// TIA Portal project "GridTest2093" (V19)

(* hardware
DEVICE "S7-1200 station_1"  S7-1200 Station
   slot 0: "Rack_0"  S7-1200 Rack  Rack  V1.0
   slot 1: "PLC_1"  CPU 1214C DC/DC/DC  6ES7 214-1AG40-0XB0  V4.6
   slot 2: "AI 4x13BIT_1"  6ES7 231-4HD32-0XB0  V2.1
   slot 3: "AI 8x13BIT_1"  6ES7 231-4HF32-0XB0  V2.1
   slot 4: "AQ 4x14BIT_1"  6ES7 232-4HD32-0XB0  V2.1
   slot 5: "DQ 8x24VDC _1"  SM 1222 DQ8 x 24VDC  6ES7 222-1BF32-0XB0  V2.0
*)

// ===== PLC "PLC_1"  CPU 1214C DC/DC/DC =====

VAR_GLOBAL   // PLC tag table "Default tag table"
   "test1" AT %Q0.0 : Bool;
   "test2" AT %Q0.1 : Bool;
END_VAR

VAR_GLOBAL   // PLC tag table "Grid"
   "o_G1_Inverter_ON" AT %Q0.2 : Bool;
   "o_G1_KV_ON" AT %Q0.3 : Bool;
   "o_G2_Inverter_ON" AT %Q0.4 : Bool;
   "o_G2_KV_ON" AT %Q0.5 : Bool;
   "ao_G1_KV_SET" AT %QW112 : Int;
   "ao_G2_KV_SET" AT %QW114 : Int;
   "ai_G1_KVFB" AT %IW96 : Int;
   "ai_G2_KVFB" AT %IW98 : Int;
END_VAR

VAR_GLOBAL   // PLC tag table "remVals"
   "ai_remKVrdg" AT %IW112 : Int;
   "ai_remMArdg" AT %IW114 : Int;
   "ai_remIfrdg" AT %IW116 : Int;
   "i_remProcOK" AT %I0.0 : Bool;
   "i_rem_NotUsed" AT %I0.1 : Bool;
   "i_cam_EXPOSE_OK" AT %I0.2 : Bool;
   "o_GoRemote" AT %Q20.0 : Bool;
   "o_remSmall" AT %Q20.1 : Bool;
   "o_remHiSpd" AT %Q20.2 : Bool;
   "o_remNotUsed" AT %Q20.3 : Bool;
   "o_Sonalert" AT %Q20.4 : Bool;
   "o_cam_SHORT_SYNC" AT %Q20.5 : Bool;
   "o_cam_LONG_SYNC" AT %Q20.6 : Bool;
   "ao_KVSP" AT %QW116 : Int;
END_VAR

DATA_BLOCK "Inputs_DB"   // DB9
{ S7_Optimized_Access := 'TRUE' }
VERSION : 0.1
// stored: InstanceOfName Inputs
"Inputs"
BEGIN
END_DATA_BLOCK

DATA_BLOCK "Step_Values_DB"   // DB16
{ S7_Optimized_Access := 'TRUE' }
VERSION : 0.1
// stored: InstanceOfName Step_Values
"Step_Values"
BEGIN
END_DATA_BLOCK

DATA_BLOCK "Outputs_DB"   // DB17
{ S7_Optimized_Access := 'TRUE' }
VERSION : 0.1
// stored: InstanceOfName Outputs
"Outputs"
BEGIN
END_DATA_BLOCK

DATA_BLOCK "Run_Sched_DB"   // DB37
{ S7_Optimized_Access := 'TRUE' }
VERSION : 0.1
// stored: InstanceOfName Run_Sched
"Run_Sched"
BEGIN
END_DATA_BLOCK

DATA_BLOCK "ALARMS_CHECK_DB"   // DB38
{ S7_Optimized_Access := 'TRUE' }
VERSION : 0.1
// stored: InstanceOfName ALARMS_CHECK
"ALARMS_CHECK"
BEGIN
END_DATA_BLOCK

DATA_BLOCK "Reset_DB"   // DB41
{ S7_Optimized_Access := 'TRUE' }
VERSION : 0.1
// stored: InstanceOfName Reset
"Reset"
BEGIN
END_DATA_BLOCK

DATA_BLOCK "Heat_Int_DB"   // DB42
{ S7_Optimized_Access := 'TRUE' }
VERSION : 0.1
// stored: InstanceOfName Heat_Int
"Heat_Int"
BEGIN
END_DATA_BLOCK

DATA_BLOCK "Retests_DB"   // DB43
{ S7_Optimized_Access := 'TRUE' }
VERSION : 0.1
// stored: InstanceOfName Retests
"Retests"
BEGIN
END_DATA_BLOCK

// folder: Datablocks

DATA_BLOCK "LVtest"   // DB1
{ S7_Optimized_Access := 'FALSE' }
VERSION : 0.1
   VAR
      val1 : Bool := false;
      val2 : Bool;
      num1 : DInt := 10;
      str1 : String := 'hello';
      val3 : Bool := false;
      str2 : String := 'nice';
      val4 : Bool;
      steptest : Int;
   END_VAR
BEGIN
END_DATA_BLOCK

DATA_BLOCK "BIASDIFF"   // DB3
{ S7_Optimized_Access := 'FALSE' }
VERSION : 0.1
   VAR
      BIAS_ZERO : Bool;
      DIFF_ZERO : Bool;
      BIAS : Real;
      DIFF : Real;
      BIAS_DIFF_OK : Bool;
      BIAS_RSE : Bool;
      BIAS_LWR : Bool;
      DIFF_RSE : Bool;
      DIFF_LWR : Bool;
      Max_DIFF : Real;
      Min_DIFF : Real;
      DIFF_TOGGLE : Bool;
      BIAS_DIFF_TMR : Time;
      BIAS_Prior : Real;
      DIFF_Prior : Real;
      delta_BIAS : Real;
   END_VAR
BEGIN
END_DATA_BLOCK

DATA_BLOCK "Gx"   // DB4
{ S7_Optimized_Access := 'FALSE' }
VERSION : 0.1
   VAR
      max_Gx : Real;
      min_Gx : Real;
      G1V_SP : Real;
      G2V_SP : Real;
      schd_max_Gx : Array[0..2] of Real;
      G1Invert : Bool;   // G1 Invert output
      G1KVOn : Bool;   // G1 KV enable output
      G1KVSet : Real;   // G1 KV set output
      G2Invert : Bool;   // G2 Invert output
      G2KVON : Bool;   // G2 KV enable output
      G2KVSet : Real;   // G2 KV set output
      G1KVfb : DInt;   // G1 KV feedback input
      G2KVfb : DInt;   // G2 KV feedback input
      Gx_LIMIT : Real;
   END_VAR
BEGIN
END_DATA_BLOCK

DATA_BLOCK "Params"   // DB5
{ S7_Optimized_Access := 'FALSE' }
VERSION : 0.1
   VAR
      stp_PARAMS : Array[0..31] of Bool;
      PARAMS : Array[0..31] of Bool;
      stp_TEST : Array[0..31] of Bool;
   END_VAR
BEGIN
END_DATA_BLOCK

DATA_BLOCK "Limits"   // DB6
{ S7_Optimized_Access := 'FALSE' }
VERSION : 0.1
   VAR
      LIMITS : Array[0..39] of Real;
      LIMITS_PB : Array[0..7] of Bool;
   END_VAR
BEGIN
   // LIMITS[0] : max GxV
   // LIMITS[1] : max GxuA
   // LIMITS[2] : max EfDr
   // LIMITS[3] : min EfDr
   // LIMITS[4] : max KV
   // LIMITS[5] : MA%HI Circ Brkr ABORT
   // LIMITS[6] : max MA ABORT
   // LIMITS[7] : GRID Comms bad mS ABORT
   // LIMITS[8] : max short pulse tries
   // LIMITS[9] : .....
   // LIMITS[10] : short EXP Cool delay mS to next
   // LIMITS[11] : mS rdg delay
   // LIMITS[12] : max Temp ABORT
   // LIMITS[13] : pulse MA OK%tol
   // LIMITS[14] : pulse If OK %tol
   // LIMITS[15] : ......
   // LIMITS[16] : EfDr delta max adj
   // LIMITS[17] : MA REG Gain
   // LIMITS[18] : If REG Gain
   // LIMITS[19] : Cutoff Test BIAS Gain
   // LIMITS[20] : If rdgs averaged
   // LIMITS[21] : MA rdgs avgd for Cutoff
   // LIMITS[22] : Xpos Offset mm
   // LIMITS[23] : Zpos Offset mm
   // LIMITS[24] : Ypos Offset mm
   // LIMITS[25] : .....
   // LIMITS[26] : .....
   // LIMITS[27] : DEFL adj Gain, V/mm LO
   // LIMITS[28] : .....
   // LIMITS[29] : Change Mode TD mS
   // LIMITS[30] : .....
   // LIMITS[31] : Heat/to TEMP params[1]
   // LIMITS[32] : Cool/to TEMP params[5]
   // LIMITS[35] : min -delta BIAS adj Width
   // LIMITS[39] : auto re-TEST # times
   // LIMITS[38] : MA REG Gain #2
   // LIMITS[37] : Width adj BIAS Gain (140KV)
   // LIMITS[36] : .....
   // LIMITS[34] : max +delta BIAS adj Width
   // LIMITS[33] : .....
   // LIMITS_PB[0] : NO GRID TANK
   // LIMITS_PB[1] : NO CAMERA
   // LIMITS_PB[2] : Cheat ProcNOK
   // LIMITS_PB[3] : SIM IO
   // LIMITS_PB[4] : store IMAGE
   // LIMITS_PB[5] : cycle Go User Sync
   // LIMITS_PB[6] : CAL (Remote = On)
   // LIMITS_PB[7] : Over Expose Alarm
END_DATA_BLOCK

DATA_BLOCK "Schd"   // DB7
{ S7_Optimized_Access := 'TRUE' }
VERSION : 0.1
   VAR
      RUN : Bool;
   END_VAR
BEGIN
END_DATA_BLOCK

DATA_BLOCK "ANALOG_IO"   // DB8
{ S7_Optimized_Access := 'FALSE' }
VERSION : 0.1
   VAR
      remKVSP : Real := 0.0;
      remKVrdg : Real := 0.0;
      remMASP : Real := 0.0;
      remMArdg : Real := 0.0;
      remEfDrSP : Real := 0.0;
      remEfDrRdg : Real := 0.0;
      remIfrdg : Real := 0.0;
      G1V_SP : Real := 0.0;
      G2V_SP : Real := 0.0;
      G1RDG : Real := 0.0;
      G2RDG : Real := 0.0;
   END_VAR
BEGIN
END_DATA_BLOCK

DATA_BLOCK "Schedule"   // DB10
{ S7_Optimized_Access := 'FALSE' }
VERSION : 0.1
   VAR
      PARAMS : Array[0..31] of Real;
      KV : Array[0..31] of Real;
      MAIF : Array[0..31] of Real;
      EXPtime : Array[0..31] of Real;
      COOLtime : Array[0..31] of Real;
      scansMode : Array[0..31] of Real;
      dataitem : Array[0..31] of Real;
      min : Array[0..31] of Real;
      max : Array[0..31] of Real;
      initBIAS : Array[0..31] of Real;
      initDIFF : Array[0..31] of Real;
      maxGx : Array[0..31] of Real;
      initEfDr : Array[0..31] of Real;
      maxTries : Array[0..31] of Real;
      TEST : Array[0..31] of Real;
      LIM1 : Array[0..31] of Real;
      LIM2 : Array[0..31] of Real;
      LIM3 : Array[0..31] of Real;
      LIM4 : Array[0..31] of Real;
   END_VAR
BEGIN
END_DATA_BLOCK

DATA_BLOCK "DIGITAL_IO"   // DB11
{ S7_Optimized_Access := 'FALSE' }
VERSION : 0.1
   VAR
      GORemote : Bool;
      remSMALL : Bool;
      remHiSpd : Bool;
      Sonalert : Bool;
      cam_SHORT_SYNC : Bool;
      cam_LONG_SYNC : Bool;
      remProcOK : Bool;
      cam_EXPOSURE_OK : Bool;
      G1V_Invert : Bool;
      G1V_On : Bool;
      G2V_Invert : Bool;
      G2V_On : Bool;
      SPARE1 : Bool;
      SPARE2 : Bool;
      SPARE3 : Bool;
      SPARE4 : Bool;
   END_VAR
BEGIN
END_DATA_BLOCK

DATA_BLOCK "OffsetGain"   // DB12
{ S7_Optimized_Access := 'FALSE' }
VERSION : 0.1
   VAR
      remKVSPOffset : Real;
      remKVSPGain : Real;
      remKVrdgOffset : Real;
      remKVrdgGain : Real;
      remMASPOffset : Real;
      remMASPGain : Real;
      remMArdgOffset : Real;
      remMArdgGain : Real;
      remEfDrSPOffset : Real;
      remEfDrSPGain : Real;
      remEfDrRdgOffset : Real;
      remEfDrRdgGain : Real;
      remIfRdgOffset : Real;
      remIfRdgGain : Real;
      G1V_SP_Offset : Real;
      G1V_SP_Gain : Real;
      G1V_RDG_Offset : Real;
      G1V_RDG_Gain : Real;
      G2V_SP_Offset : Real;
      G2V_SP_Gain : Real;
      G2V_RDG_Offset : Real;
      G2V_RDG_Gain : Real;
   END_VAR
BEGIN
END_DATA_BLOCK

DATA_BLOCK "Tube"   // DB13
{ S7_Optimized_Access := 'FALSE' }
VERSION : 0.1
   VAR
      RTC : Real;
      HS : Real;
      T100 : Real;
      T0 : Real;
      AP : Real;
   END_VAR
BEGIN
END_DATA_BLOCK

DATA_BLOCK "Run_Control"   // DB14
{ S7_Optimized_Access := 'FALSE' }
VERSION : 0.1
   VAR
      First_Step : Int;
      Final_Step : Int;
      Current_Step : Int;
      Run : Int;
      Reset : Int;
      GoRemote : Int;
   END_VAR
BEGIN
END_DATA_BLOCK

DATA_BLOCK "Alarms"   // DB15
{ S7_Optimized_Access := 'FALSE' }
VERSION : 0.1
   VAR
      Alarms : Array[0..31] of Bool;
      Alarm_Clear : Bool;
      buff1 : Int;
      ProcNOK_Clear : Bool;
      buff2 : Int;
      ALARM_ACTIVE : Bool;
      PROCNOK_ACTIVE : Bool;
   END_VAR
BEGIN
   // Alarms[0] : COMMS ERROR
   // Alarms[1] : RUN LOG OPEN >> CLOSE
   // Alarms[2] : remProcNOK 50 sec
   // Alarms[3] : expose NOK 90 sec
   // Alarms[4] : exp NOK 5min >> ABORT
   // Alarms[5] : GRID COMMS >> ABORT
   // Alarms[6] : MA HI >> ABORT
   // Alarms[7] : max tries LIM[9] >> ABORT
   // Alarms[8] : ProcNOK 90 sec
   // Alarms[9] : ProcNOK CHEATED (LIM)
   // Alarms[10] : Gx Volts HI/LO
   // Alarms[11] : TEMP HI LIM[13] >> ABORT
   // Alarms[12] : Cam User Sync <> 2 15 sec
   // Alarms[13] : CLOSE DATA SHEET LOG
   // Alarms[14] : Gx uA > LIM[2] >> ABORT
   // Alarms[15] : EXPOSE LONG >> ABORT
   // Alarms[31] : DONE
END_DATA_BLOCK

DATA_BLOCK "Cam"   // DB18
{ S7_Optimized_Access := 'FALSE' }
VERSION : 0.1
   VAR
      X_defl : Real;
      Z_defl : Real;
      Y_defl : Real;
      cam_Wref : Real;
      cam_Lref : Real;
      cam_Xref : Real;
      cam_Zref : Real;
      cam_Yref : Real;
      cam_WIDTH : Real;
      cam_LENGTH : Real;
      cam_Xpos : Real;
      cam_Zpos : Real;
      cam_Ypos : Real;
      cam_MAG : Real;
      cam_FRAME_RATE : Real;
      image_KV : Real;
      image_MA : Real;
      image_G1 : Real;
      image_G2 : Real;
      image_BIAS : Real;
      image_DIFF : Real;
      cam_POS : Real;
      cam_USER_SYNC : Int;
      cam_DATA : Int;
      BIAS_ref : Int;
      cam_PEAK : Int;
      cam_OB_pk : Int;
      cam_Mode : Int;
      cam_PERCENT_MAX : Int;
      NO_CAMERA : Bool;
      IMAGE_ACQUIRED : Bool;
      STORE_IMAGE : Bool;
      cam_CAL_OFFSET : Bool;
      cam_STATUS : String;
      cam_IMAGE_PATH : String;
   END_VAR
BEGIN
END_DATA_BLOCK

DATA_BLOCK "pulse"   // DB19
{ S7_Optimized_Access := 'TRUE' }
VERSION : 0.1
   VAR
      pulse_KV : Int;
      pulse_MA : Int;
      pulse_If : Int;
      pulse_EfDr : Int;
      pulse_G2 : Int;
      pulse_G1 : Int;
      shortpulse_tries : Int;
      XPOSE_SEC : Int;
      COOL_SEC : Int;
      rdgs_avgd : Int;
      shortpulsetmr : Time;
      pulsePeriod : Real;
   END_VAR
BEGIN
END_DATA_BLOCK

DATA_BLOCK "ref"   // DB20
{ S7_Optimized_Access := 'TRUE' }
VERSION : 0.1
   VAR
      EfDr_ref : Real;
      BIAS_ref : Real;
   END_VAR
BEGIN
END_DATA_BLOCK

DATA_BLOCK "Prior"   // DB21
{ S7_Optimized_Access := 'TRUE' }
VERSION : 0.1
   VAR
      BIAS_Prior : Real;
      DIFF_Prior : Real;
      EfDr_Prior : Real;
   END_VAR
BEGIN
END_DATA_BLOCK

DATA_BLOCK "Results"   // DB22
{ S7_Optimized_Access := 'FALSE' }
VERSION : 0.1
   VAR
      testVAL : Real;
      min : Real;
      max : Real;
      KV : Real;
      MA : Real;
      EfDr : Real;
      "If" : Real;
      Temp : Real;
      G1V : Real;
      G2V : Real;
      Width : Real;
      Length : Real;
      Xdefl : Real;
      Zdefl : Real;
      Ydefl : Real;
      Xpos : Real;
      Zpos : Real;
      Ypos : Real;
      Mag : Real;
      pk : Real;
      OBpk : Real;
      tries : Real;
      scansmode : Real;
      dataitem : Real;
      Pass_Fail : Int;
   END_VAR
BEGIN
END_DATA_BLOCK

DATA_BLOCK "Chain_Schedule"   // DB23
{ S7_Optimized_Access := 'TRUE' }
VERSION : 0.1
   VAR
      Params : Real;
      KV : Real;
      MAIf : Real;
      EXPtime : Real;
      COOLtime : Real;
      scansMode : Real;
      dataitem : Real;
      min : Real;
      max : Real;
      initBIAS : Real;
      initDIFF : Real;
      maxGx : Real;
      initEfDr : Real;
      maxTries : Real;
      TEST : Real;
      LIM1 : Real;
      LIM2 : Real;
      LIM3 : Real;
      LIM4 : Real;
   END_VAR
BEGIN
END_DATA_BLOCK

DATA_BLOCK "System"   // DB24
{ S7_Optimized_Access := 'FALSE' }
VERSION : 0.1
   VAR
      COOLING : Bool;
      GoRemote : Bool;
      Temp_set : Real;
      Temp_rdg : Real;
      XPOSE_SEC : Real;
      RPTS : Int;
      Exp_MA_If_OK : Bool;
      Sleep : Bool;
   END_VAR
BEGIN
END_DATA_BLOCK

DATA_BLOCK "ProcOK"   // DB25
{ S7_Optimized_Access := 'FALSE' }
VERSION : 0.1
   VAR
      ProcOKArray : Array[0..31] of Bool;
      ProcOK : Bool;
   END_VAR
BEGIN
   ProcOKArray[0] := true;
   ProcOKArray[1] := true;
   ProcOKArray[2] := true;
   ProcOKArray[3] := true;
   ProcOKArray[4] := true;
   ProcOKArray[5] := true;
   ProcOKArray[6] := true;
   ProcOKArray[7] := true;
   ProcOKArray[8] := true;
   ProcOKArray[9] := true;
   ProcOKArray[10] := true;
   ProcOKArray[11] := true;
   ProcOKArray[12] := true;
   ProcOKArray[13] := true;
   ProcOKArray[14] := true;
   ProcOKArray[15] := true;
   ProcOKArray[16] := true;
   ProcOKArray[17] := true;
   ProcOKArray[18] := true;
   ProcOKArray[19] := true;
   ProcOKArray[20] := true;
   ProcOKArray[21] := true;
   ProcOKArray[22] := true;
   ProcOKArray[23] := true;
   ProcOKArray[24] := true;
   ProcOKArray[25] := true;
   ProcOKArray[26] := true;
   ProcOKArray[27] := true;
   ProcOKArray[28] := true;
   ProcOKArray[29] := true;
   ProcOKArray[30] := true;
   ProcOKArray[31] := true;
END_DATA_BLOCK

DATA_BLOCK "StepVals"   // DB26
{ S7_Optimized_Access := 'TRUE' }
VERSION : 0.1
   VAR
      PARAMS : Real;
      KV : Real;
      MAIf : Real;
      EXPtime : Real;
      COOLtime : Real;
      scansMode : Real;
      dataitem : Real;
      min : Real;
      max : Real;
      initBIAS : Real;
      initDIFF : Real;
      maxGx : Real;
      initEfDr : Real;
      maxTries : Real;
      TEST : Real;
      LIM1 : Real;
      LIM2 : Real;
      LIM3 : Real;
      LIM4 : Real;
   END_VAR
BEGIN
END_DATA_BLOCK

DATA_BLOCK "Misc"   // DB31
{ S7_Optimized_Access := 'FALSE' }
VERSION : 0.1
   VAR
      CutOff_avg_MA : Bool;
      rem_MA_rdg_avg : Real;
      Blinkingtme : Real;
   END_VAR
BEGIN
END_DATA_BLOCK

DATA_BLOCK "Cutoff"   // DB32
{ S7_Optimized_Access := 'TRUE' }
VERSION : 0.1
   VAR
      cutoff_BIAS : Real;
      cutoff_avg_MA : Bool;
   END_VAR
BEGIN
END_DATA_BLOCK

DATA_BLOCK "Remote"   // DB33
{ S7_Optimized_Access := 'TRUE' }
VERSION : 0.1
   VAR
      remEfDr_SP : Real;
   END_VAR
BEGIN
END_DATA_BLOCK

DATA_BLOCK "Cam(int)"   // DB34
{ S7_Optimized_Access := 'FALSE' }
VERSION : 0.1
   VAR
      cam_USER_SYNC : Int;
      cam_DATA : Int;
      BIAS_ref : Int;
      cam_PEAK : Int;
      cam_OB_pk : Int;
      cam_Mode : Int;
      cam_PERCENT_MAX : Int;
   END_VAR
BEGIN
END_DATA_BLOCK

DATA_BLOCK "Cam(bool)"   // DB35
{ S7_Optimized_Access := 'FALSE' }
VERSION : 0.1
   VAR
      NO_CAMERA : Bool;
      IMAGE_ACQUIRED : Bool;
      STORE_IMAGE : Bool;
      cam_CAL_OFFSET : Bool;
   END_VAR
BEGIN
END_DATA_BLOCK

DATA_BLOCK "Cam(string)"   // DB36
{ S7_Optimized_Access := 'FALSE' }
VERSION : 0.1
   VAR
      cam_STATUS : String;
      cam_IMAGE_PATH : String;
   END_VAR
BEGIN
END_DATA_BLOCK

DATA_BLOCK "Process"   // DB39
{ S7_Optimized_Access := 'FALSE' }
VERSION : 0.1
   VAR
      Run_Init : Bool;
      Step_Init : Bool := true;
      Running : Bool;
      Step_Running : Bool;
      Step_Done : Bool;
      Schedule_Done : Bool;
      Retest_Done : Bool;
      Results_Ready : Bool;
   END_VAR
BEGIN
END_DATA_BLOCK

DATA_BLOCK "Retest"   // DB40
{ S7_Optimized_Access := 'FALSE' }
VERSION : 0.1
   VAR
      Retest_Step : Int;
      Retest_End : Int;
      Retest_Type : Int;   // Retest=1: Retest Retest_Step only; Retest=2: Retest Retest_Step to End
      Retests : Int;
      Retries : Int;
      Retest : Bool;
   END_VAR
BEGIN
END_DATA_BLOCK

// folder: System blocks/Program resources

DATA_BLOCK "IEC_Timer_0_DB"   // DB2
{ S7_Optimized_Access := 'FALSE' }
AUTHOR : Simatic
FAMILY : IEC
NAME : IEC_TMR
VERSION : 1.0
// stored: InstanceOfName IEC_TIMER
"IEC_TIMER"
BEGIN
END_DATA_BLOCK

DATA_BLOCK "BIAS_Step_tmr1"   // DB27
{ S7_Optimized_Access := 'TRUE' }
AUTHOR : Simatic
FAMILY : IEC
NAME : IEC_TMR
VERSION : 1.0
// stored: InstanceOfName IEC_TIMER
"IEC_TIMER"
BEGIN
END_DATA_BLOCK

DATA_BLOCK "BIAS_Step_tmr2"   // DB28
{ S7_Optimized_Access := 'TRUE' }
AUTHOR : Simatic
FAMILY : IEC
NAME : IEC_TMR
VERSION : 1.0
// stored: InstanceOfName IEC_TIMER
"IEC_TIMER"
BEGIN
END_DATA_BLOCK

DATA_BLOCK "BIAS_Step_tmr3"   // DB29
{ S7_Optimized_Access := 'TRUE' }
AUTHOR : Simatic
FAMILY : IEC
NAME : IEC_TMR
VERSION : 1.0
// stored: InstanceOfName IEC_TIMER
"IEC_TIMER"
BEGIN
END_DATA_BLOCK

DATA_BLOCK "BIAS_Step_tmr4"   // DB30
{ S7_Optimized_Access := 'TRUE' }
AUTHOR : Simatic
FAMILY : IEC
NAME : IEC_TMR
VERSION : 1.0
// stored: InstanceOfName IEC_TIMER
"IEC_TIMER"
BEGIN
END_DATA_BLOCK

// folder: (top level)

ORGANIZATION_BLOCK "Main"   // OB1, LAD, ProgramCycle
TITLE = "Main Program Sweep (Cycle)"
{ S7_Optimized_Access := 'TRUE' }
VERSION : 0.1
   VAR_INPUT
      Initial_Call : Bool;   // Initial call of this OB
      Remanence : Bool;   // =True, if remanent data are available
   END_VAR
   VAR_TEMP
      test : Bool;
      "step" : Int;
      Blinkingtimer : Real;
   END_VAR
   VAR_TEMP   // added for the SCL form of the ladder/FBD networks
      _w1 : Bool;
   END_VAR
BEGIN

REGION Network 1
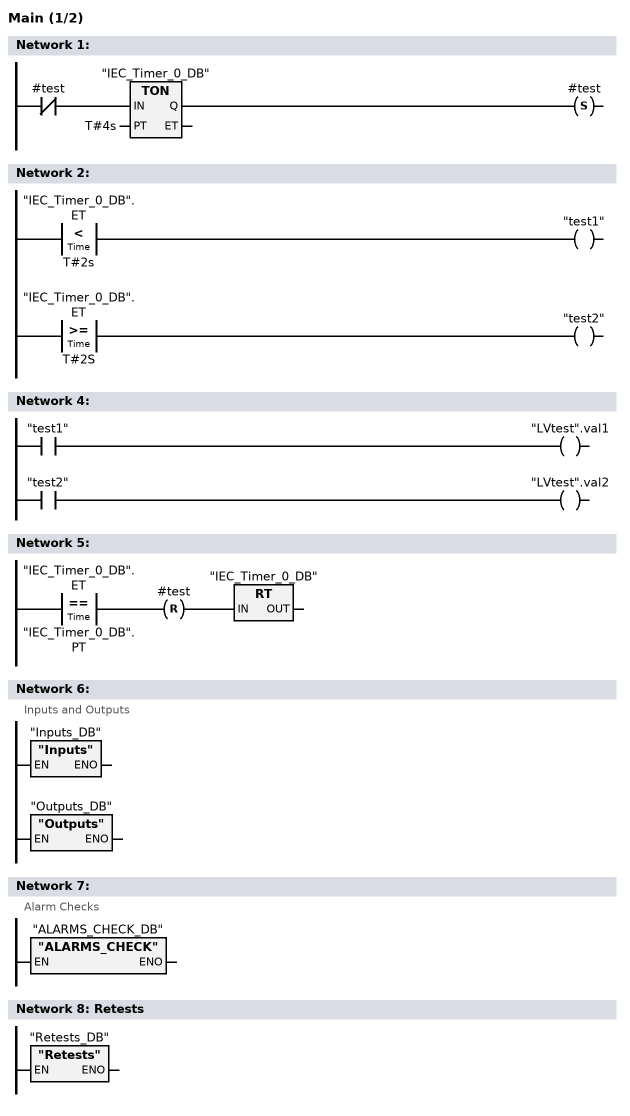
   "IEC_Timer_0_DB".TON(IN := NOT #test, PT := T#4s);
   IF "IEC_Timer_0_DB".Q THEN #test := TRUE; END_IF;
END_REGION

REGION Network 2
   RUNG wire#powerrail
      { S7_Templates := "SrcType := Time" } LT_Contact(in1 := "IEC_Timer_0_DB".ET, in2 := T#2s)
      Coil( "test1" )
   END_RUNG
   RUNG wire#powerrail
      { S7_Templates := "SrcType := Time" } GE_Contact(in1 := "IEC_Timer_0_DB".ET, in2 := T#2S)
      Coil( "test2" )
   END_RUNG
   // the same network as SCL:
   "test1" := "IEC_Timer_0_DB".ET < T#2s;
   "test2" := "IEC_Timer_0_DB".ET >= T#2S;
END_REGION

REGION Network 3 (SCL)
   "Misc".Blinkingtme := INT_TO_REAL(TIME_TO_INT("IEC_Timer_0_DB".ET));
END_REGION

REGION Network 4
   RUNG wire#powerrail
      Contact( "test1" )
      Coil( "LVtest".val1 )
   END_RUNG
   RUNG wire#powerrail
      Contact( "test2" )
      Coil( "LVtest".val2 )
   END_RUNG
   // the same network as SCL:
   "LVtest".val1 := "test1";
   "LVtest".val2 := "test2";
END_REGION

REGION Network 5
   RUNG wire#powerrail
      { S7_Templates := "SrcType := Time" } EQ_Contact(in1 := "IEC_Timer_0_DB".ET, in2 := "IEC_Timer_0_DB".PT)
      R_Coil( #test )
      RT_Coil( "IEC_Timer_0_DB" )
   END_RUNG
   // the same network as SCL:
   #_w1 := "IEC_Timer_0_DB".ET = "IEC_Timer_0_DB".PT;
   IF #_w1 THEN
       #test := FALSE;
       RESET_TIMER("IEC_Timer_0_DB");
   END_IF;
END_REGION

REGION Network 6
   // Inputs and Outputs
   RUNG wire#powerrail
      "Inputs_DB"()
   END_RUNG
   RUNG wire#powerrail
      "Outputs_DB"()
   END_RUNG
   // the same network as SCL:
   "Inputs_DB"();   // "Inputs"
   "Outputs_DB"();   // "Outputs"
END_REGION

REGION Network 7
   // Alarm Checks
   RUNG wire#powerrail
      "ALARMS_CHECK_DB"()
   END_RUNG
   // the same network as SCL:
   "ALARMS_CHECK_DB"();   // "ALARMS_CHECK"
END_REGION

REGION Network 8: Retests
   RUNG wire#powerrail
      "Retests_DB"()
   END_RUNG
   // the same network as SCL:
   "Retests_DB"();   // "Retests"
END_REGION

REGION Network 9
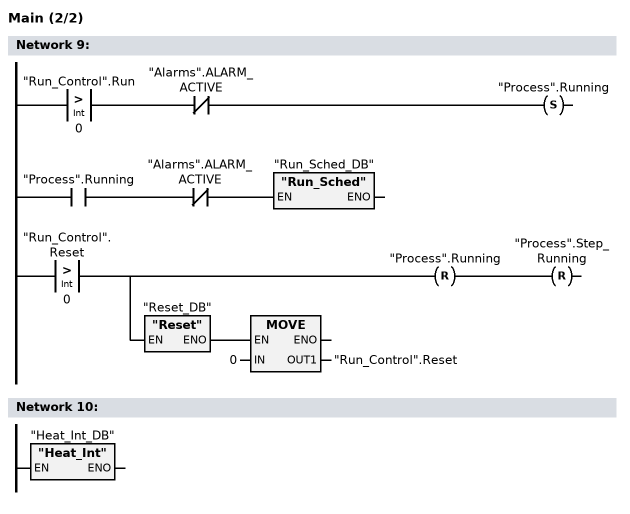
   RUNG wire#powerrail
      { S7_Templates := "SrcType := Int" } GT_Contact(in1 := "Run_Control".Run, in2 := 0)
      I_Contact( "Alarms".ALARM_ACTIVE )
      S_Coil( "Process".Running )
   END_RUNG
   RUNG wire#powerrail
      Contact( "Process".Running )
      I_Contact( "Alarms".ALARM_ACTIVE )
      "Run_Sched_DB"()
   END_RUNG
   RUNG wire#powerrail
      { S7_Templates := "SrcType := Int" } GT_Contact(in1 := "Run_Control".Reset, in2 := 0)
      wire#w1
      R_Coil( "Process".Running )
      R_Coil( "Process".Step_Running )
   END_RUNG
   RUNG wire#w1
      "Reset_DB"()
      Move(in := 0, out1 => "Run_Control".Reset)
   END_RUNG
   // the same network as SCL:
   IF ("Run_Control".Run > 0) AND NOT "Alarms".ALARM_ACTIVE THEN "Process".Running := TRUE; END_IF;
   IF "Process".Running AND NOT "Alarms".ALARM_ACTIVE THEN
       "Run_Sched_DB"();   // "Run_Sched"
   END_IF;
   IF "Run_Control".Reset > 0 THEN
       "Process".Running := FALSE;
       "Process".Step_Running := FALSE;
   END_IF;
   "Reset_DB"(EN := "Run_Control".Reset > 0, ENO => #_w1);   // "Reset"
   IF #_w1 THEN "Run_Control".Reset := 0; END_IF;
END_REGION

REGION Network 10
   RUNG wire#powerrail
      "Heat_Int_DB"()
   END_RUNG
   // the same network as SCL:
   "Heat_Int_DB"();   // "Heat_Int"
END_REGION
END_ORGANIZATION_BLOCK

ORGANIZATION_BLOCK "Startup"   // OB100, LAD, Startup
TITLE = "Complete Restart"
{ S7_Optimized_Access := 'TRUE' }
VERSION : 0.1
   VAR_INPUT
      LostRetentive : Bool;   // True if retentive data are lost
      LostRTC : Bool;   // True if date and time are lost
   END_VAR
BEGIN
END_ORGANIZATION_BLOCK

// folder: Main Routine

FUNCTION_BLOCK "BIAS DIFF"   // FB1, LAD
{ S7_Optimized_Access := 'TRUE' }
VERSION : 0.1
   VAR
      BIAS_DIFF_TMR : TON_TIME;
   END_VAR
BEGIN

REGION Network 1 (SCL): Set max and min Gx voltage values.
   IF "Run_Control".Run > 0 THEN
       "Gx".max_Gx := "Schedule".maxGx["Run_Control".Current_Step];
   ELSE
       "Gx".max_Gx := "Limits".LIMITS[1-1];
   END_IF;

   "Gx".min_Gx := 0;
END_REGION

REGION Network 2: Clamp BIAS to 0.0 and max_Gx
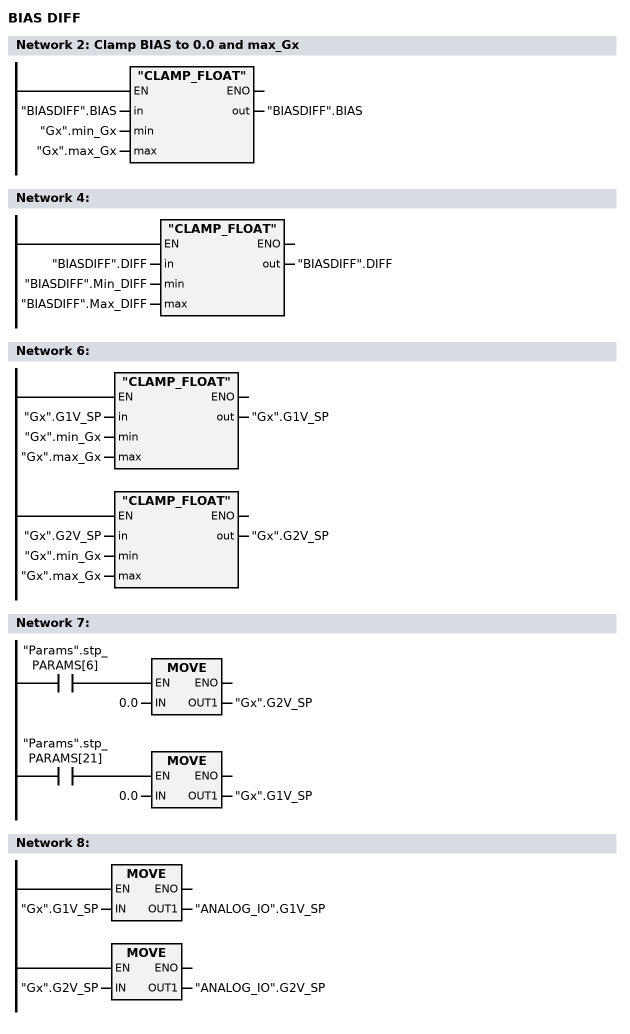
   RUNG wire#powerrail
      "CLAMP_FLOAT"(in := "BIASDIFF".BIAS, min := "Gx".min_Gx, max := "Gx".max_Gx, out => "BIASDIFF".BIAS)
   END_RUNG
   // the same network as SCL:
   "CLAMP_FLOAT"(in := "BIASDIFF".BIAS, min := "Gx".min_Gx, max := "Gx".max_Gx, out => "BIASDIFF".BIAS);
END_REGION

REGION Network 3 (SCL)
   "BIASDIFF".Max_DIFF := 2 * "BIASDIFF".BIAS;
   "BIASDIFF".Min_DIFF := -2 * "BIASDIFF".BIAS;
END_REGION

REGION Network 4
   RUNG wire#powerrail
      "CLAMP_FLOAT"(in := "BIASDIFF".DIFF, min := "BIASDIFF".Min_DIFF, max := "BIASDIFF".Max_DIFF, out => "BIASDIFF".DIFF)
   END_RUNG
   // the same network as SCL:
   "CLAMP_FLOAT"(in := "BIASDIFF".DIFF,
                 min := "BIASDIFF".Min_DIFF,
                 max := "BIASDIFF".Max_DIFF,
                 out => "BIASDIFF".DIFF);
END_REGION

REGION Network 5 (SCL)
   "Gx".G1V_SP := "BIASDIFF".BIAS + "BIASDIFF".DIFF / 2;
   "Gx".G2V_SP := "BIASDIFF".BIAS - "BIASDIFF".DIFF / 2;
END_REGION

REGION Network 6
   RUNG wire#powerrail
      "CLAMP_FLOAT"(in := "Gx".G1V_SP, min := "Gx".min_Gx, max := "Gx".max_Gx, out => "Gx".G1V_SP)
   END_RUNG
   RUNG wire#powerrail
      "CLAMP_FLOAT"(in := "Gx".G2V_SP, min := "Gx".min_Gx, max := "Gx".max_Gx, out => "Gx".G2V_SP)
   END_RUNG
   // the same network as SCL:
   "CLAMP_FLOAT"(in := "Gx".G1V_SP, min := "Gx".min_Gx, max := "Gx".max_Gx, out => "Gx".G1V_SP);
   "CLAMP_FLOAT"(in := "Gx".G2V_SP, min := "Gx".min_Gx, max := "Gx".max_Gx, out => "Gx".G2V_SP);
END_REGION

REGION Network 7
   RUNG wire#powerrail
      Contact( "Params".stp_PARAMS[6] )
      Move(in := 0.0, out1 => "Gx".G2V_SP)
   END_RUNG
   RUNG wire#powerrail
      Contact( "Params".stp_PARAMS[21] )
      Move(in := 0.0, out1 => "Gx".G1V_SP)
   END_RUNG
   // the same network as SCL:
   IF "Params".stp_PARAMS[6] THEN "Gx".G2V_SP := 0.0; END_IF;
   IF "Params".stp_PARAMS[21] THEN "Gx".G1V_SP := 0.0; END_IF;
END_REGION

REGION Network 8
   RUNG wire#powerrail
      Move(in := "Gx".G1V_SP, out1 => "ANALOG_IO".G1V_SP)
   END_RUNG
   RUNG wire#powerrail
      Move(in := "Gx".G2V_SP, out1 => "ANALOG_IO".G2V_SP)
   END_RUNG
   // the same network as SCL:
   "ANALOG_IO".G1V_SP := "Gx".G1V_SP;
   "ANALOG_IO".G2V_SP := "Gx".G2V_SP;
END_REGION
END_FUNCTION_BLOCK

FUNCTION_BLOCK "Inputs"   // FB2, LAD
{ S7_Optimized_Access := 'TRUE' }
VERSION : 0.1
BEGIN

REGION Network 1: GxV Readings
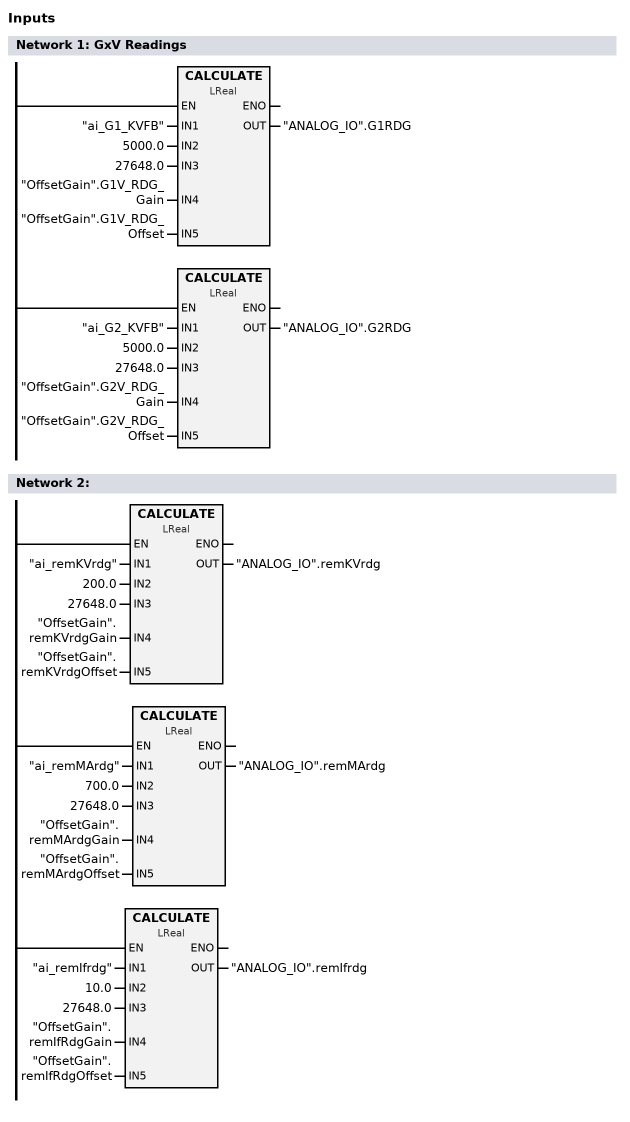
   RUNG wire#powerrail
      { S7_Templates := "SrcType := LReal"; S7_Expression := "(IN2 * IN1) / IN3 * IN4 + (IN2*IN5)" } Calculate(in1 := "ai_G1_KVFB", in2 := 5000.0, in3 := 27648.0, in4 := "OffsetGain".G1V_RDG_Gain, in5 := "OffsetGain".G1V_RDG_Offset, out => "ANALOG_IO".G1RDG)
   END_RUNG
   RUNG wire#powerrail
      { S7_Templates := "SrcType := LReal"; S7_Expression := "(IN2 * IN1) / IN3 * IN4 + (IN2*IN5)" } Calculate(in1 := "ai_G2_KVFB", in2 := 5000.0, in3 := 27648.0, in4 := "OffsetGain".G2V_RDG_Gain, in5 := "OffsetGain".G2V_RDG_Offset, out => "ANALOG_IO".G2RDG)
   END_RUNG
   // the same network as SCL:
   "ANALOG_IO".G1RDG := (5000.0 * "ai_G1_KVFB") / 27648.0 * "OffsetGain".G1V_RDG_Gain + (5000.0*"OffsetGain".G1V_RDG_Offset);
   "ANALOG_IO".G2RDG := (5000.0 * "ai_G2_KVFB") / 27648.0 * "OffsetGain".G2V_RDG_Gain + (5000.0*"OffsetGain".G2V_RDG_Offset);
END_REGION

REGION Network 2
   RUNG wire#powerrail
      { S7_Templates := "SrcType := LReal"; S7_Expression := "(IN2 * IN1) / IN3 * IN4 + (IN2*IN5)" } Calculate(in1 := "ai_remKVrdg", in2 := 200.0, in3 := 27648.0, in4 := "OffsetGain".remKVrdgGain, in5 := "OffsetGain".remKVrdgOffset, out => "ANALOG_IO".remKVrdg)
   END_RUNG
   RUNG wire#powerrail
      { S7_Templates := "SrcType := LReal"; S7_Expression := "(IN2 * IN1) / IN3 * IN4 + (IN2*IN5)" } Calculate(in1 := "ai_remMArdg", in2 := 700.0, in3 := 27648.0, in4 := "OffsetGain".remMArdgGain, in5 := "OffsetGain".remMArdgOffset, out => "ANALOG_IO".remMArdg)
   END_RUNG
   RUNG wire#powerrail
      { S7_Templates := "SrcType := LReal"; S7_Expression := "(IN2 * IN1) / IN3 * IN4 + (IN2*IN5)" } Calculate(in1 := "ai_remIfrdg", in2 := 10.0, in3 := 27648.0, in4 := "OffsetGain".remIfRdgGain, in5 := "OffsetGain".remIfRdgOffset, out => "ANALOG_IO".remIfrdg)
   END_RUNG
   // the same network as SCL:
   "ANALOG_IO".remKVrdg := (200.0 * "ai_remKVrdg") / 27648.0 * "OffsetGain".remKVrdgGain + (200.0*"OffsetGain".remKVrdgOffset);
   "ANALOG_IO".remMArdg := (700.0 * "ai_remMArdg") / 27648.0 * "OffsetGain".remMArdgGain + (700.0*"OffsetGain".remMArdgOffset);
   "ANALOG_IO".remIfrdg := (10.0 * "ai_remIfrdg") / 27648.0 * "OffsetGain".remIfRdgGain + (10.0*"OffsetGain".remIfRdgOffset);
END_REGION
END_FUNCTION_BLOCK

FUNCTION_BLOCK "Outputs"   // FB3, LAD
{ S7_Optimized_Access := 'TRUE' }
VERSION : 0.1
BEGIN

REGION Network 1: GxV Setpoints
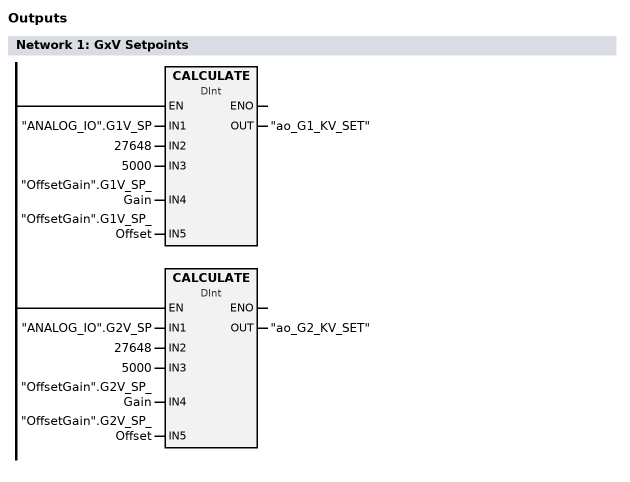
   RUNG wire#powerrail
      { S7_Templates := "SrcType := DInt"; S7_Expression := "(IN1 * IN2 * IN4 / IN3) + (IN2 * IN5)" } Calculate(in1 := "ANALOG_IO".G1V_SP, in2 := 27648, in3 := 5000, in4 := "OffsetGain".G1V_SP_Gain, in5 := "OffsetGain".G1V_SP_Offset, out => "ao_G1_KV_SET")
   END_RUNG
   RUNG wire#powerrail
      { S7_Templates := "SrcType := DInt"; S7_Expression := "(IN1 * IN2 * IN4 / IN3) + (IN2 * IN5)" } Calculate(in1 := "ANALOG_IO".G2V_SP, in2 := 27648, in3 := 5000, in4 := "OffsetGain".G2V_SP_Gain, in5 := "OffsetGain".G2V_SP_Offset, out => "ao_G2_KV_SET")
   END_RUNG
   // the same network as SCL:
   "ao_G1_KV_SET" := ("ANALOG_IO".G1V_SP * 27648 * "OffsetGain".G1V_SP_Gain / 5000) + (27648 * "OffsetGain".G1V_SP_Offset);
   "ao_G2_KV_SET" := ("ANALOG_IO".G2V_SP * 27648 * "OffsetGain".G2V_SP_Gain / 5000) + (27648 * "OffsetGain".G2V_SP_Offset);
END_REGION

REGION Network 2: Remote Setpoints
END_REGION
END_FUNCTION_BLOCK

FUNCTION_BLOCK "Step_Values"   // FB5, LAD
{ S7_Optimized_Access := 'TRUE' }
VERSION : 0.1
   VAR_INPUT
      Step_Input : Int;
   END_VAR
   VAR
      "BIAS DIFF_Instance" : "BIAS DIFF";
   END_VAR
   VAR_TEMP
      "step" : Int;
   END_VAR
   VAR_TEMP   // added for the SCL form of the ladder/FBD networks
      _w1 : Bool;
   END_VAR
BEGIN

REGION Network 1 (SCL): Move schedule values into the run variables.
   #step := #Step_Input - 1;


   "StepVals".PARAMS := "Schedule".PARAMS[#step];
   "StepVals".KV := "Schedule".KV[#step];
   "StepVals".MAIf := "Schedule".MAIF[#step];
   "StepVals".EXPtime := "Schedule".EXPtime[#step];
   "StepVals".COOLtime := "Schedule".COOLtime[#step];
   "StepVals".scansMode := "Schedule".scansMode[#step];
   "StepVals".dataitem := "Schedule".dataitem[#step];
   "StepVals".min := "Schedule".min[#step];
   "StepVals".max := "Schedule".max[#step];
   "StepVals".initBIAS := "Schedule".initBIAS[#step];
   "StepVals".initDIFF := "Schedule".initDIFF[#step];
   "StepVals".maxGx := "Schedule".maxGx[#step];
   "StepVals".initEfDr := "Schedule".initEfDr[#step];
   "StepVals".maxTries := "Schedule".maxTries[#step];
   "StepVals".TEST := "Schedule".TEST[#step];
   "StepVals".LIM1 :="Schedule".LIM1[#step];
   "StepVals".LIM2 := "Schedule".LIM2[#step];
   "StepVals".LIM3 := "Schedule".LIM3[#step];
   "StepVals".LIM4 := "Schedule".LIM4[#step];
END_REGION

REGION Network 2: Decode step PARAMS and TEST
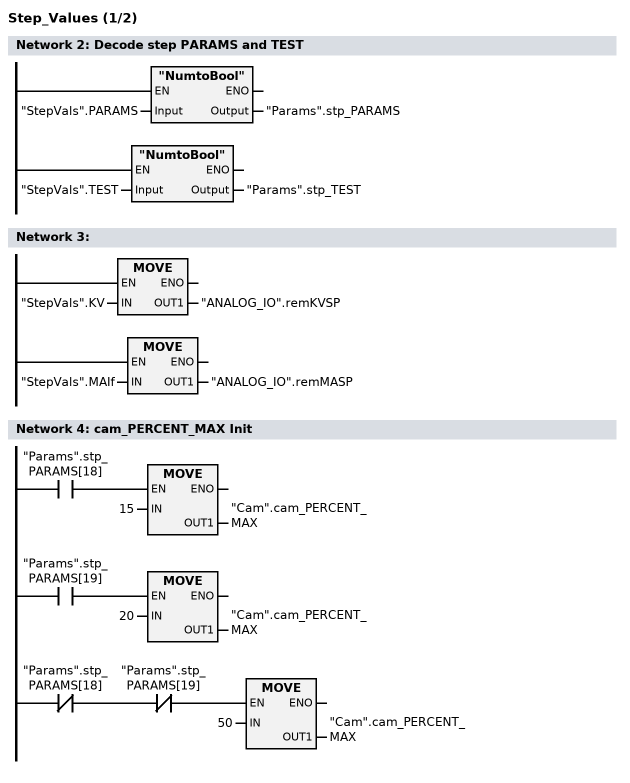
   RUNG wire#powerrail
      "NumtoBool"(Input := "StepVals".PARAMS, Output => "Params".stp_PARAMS)
   END_RUNG
   RUNG wire#powerrail
      "NumtoBool"(Input := "StepVals".TEST, Output => "Params".stp_TEST)
   END_RUNG
   // the same network as SCL:
   "NumtoBool"(Input := "StepVals".PARAMS, Output => "Params".stp_PARAMS);
   "NumtoBool"(Input := "StepVals".TEST, Output => "Params".stp_TEST);
END_REGION

REGION Network 3
   RUNG wire#powerrail
      Move(in := "StepVals".KV, out1 => "ANALOG_IO".remKVSP)
   END_RUNG
   RUNG wire#powerrail
      Move(in := "StepVals".MAIf, out1 => "ANALOG_IO".remMASP)
   END_RUNG
   // the same network as SCL:
   "ANALOG_IO".remKVSP := "StepVals".KV;
   "ANALOG_IO".remMASP := "StepVals".MAIf;
END_REGION

REGION Network 4: cam_PERCENT_MAX Init
   RUNG wire#powerrail
      Contact( "Params".stp_PARAMS[18] )
      Move(in := 15, out1 => "Cam".cam_PERCENT_MAX)
   END_RUNG
   RUNG wire#powerrail
      Contact( "Params".stp_PARAMS[19] )
      Move(in := 20, out1 => "Cam".cam_PERCENT_MAX)
   END_RUNG
   RUNG wire#powerrail
      I_Contact( "Params".stp_PARAMS[18] )
      I_Contact( "Params".stp_PARAMS[19] )
      Move(in := 50, out1 => "Cam".cam_PERCENT_MAX)
   END_RUNG
   // the same network as SCL:
   IF "Params".stp_PARAMS[18] THEN "Cam".cam_PERCENT_MAX := 15; END_IF;
   IF "Params".stp_PARAMS[19] THEN "Cam".cam_PERCENT_MAX := 20; END_IF;
   IF NOT "Params".stp_PARAMS[18] AND NOT "Params".stp_PARAMS[19] THEN "Cam".cam_PERCENT_MAX := 50; END_IF;
END_REGION

REGION Network 5
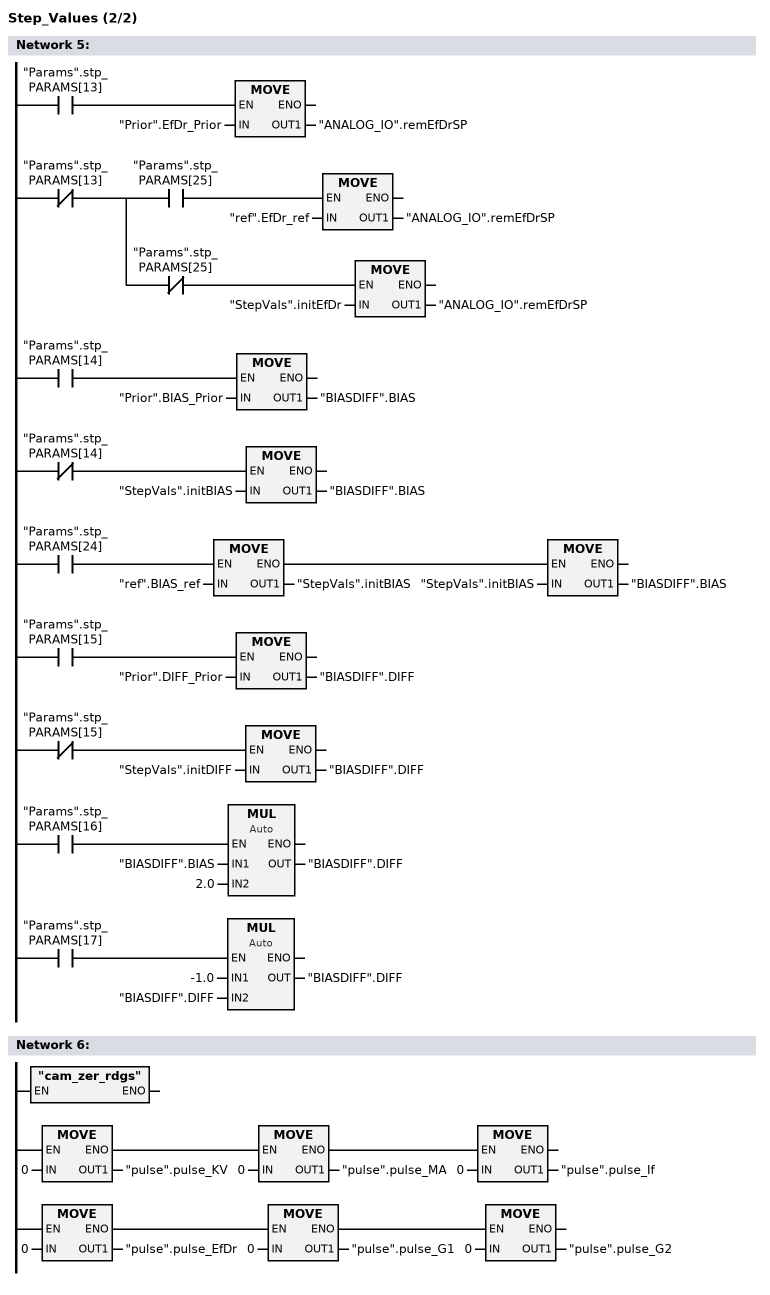
   RUNG wire#powerrail
      Contact( "Params".stp_PARAMS[13] )
      Move(in := "Prior".EfDr_Prior, out1 => "ANALOG_IO".remEfDrSP)
   END_RUNG
   RUNG wire#powerrail
      I_Contact( "Params".stp_PARAMS[13] )
      wire#w1
      Contact( "Params".stp_PARAMS[25] )
      Move(in := "ref".EfDr_ref, out1 => "ANALOG_IO".remEfDrSP)
   END_RUNG
   RUNG wire#w1
      I_Contact( "Params".stp_PARAMS[25] )
      Move(in := "StepVals".initEfDr, out1 => "ANALOG_IO".remEfDrSP)
   END_RUNG
   RUNG wire#powerrail
      Contact( "Params".stp_PARAMS[14] )
      Move(in := "Prior".BIAS_Prior, out1 => "BIASDIFF".BIAS)
   END_RUNG
   RUNG wire#powerrail
      I_Contact( "Params".stp_PARAMS[14] )
      Move(in := "StepVals".initBIAS, out1 => "BIASDIFF".BIAS)
   END_RUNG
   RUNG wire#powerrail
      Contact( "Params".stp_PARAMS[24] )
      Move(in := "ref".BIAS_ref, out1 => "StepVals".initBIAS)
      Move(in := "StepVals".initBIAS, out1 => "BIASDIFF".BIAS)
   END_RUNG
   RUNG wire#powerrail
      Contact( "Params".stp_PARAMS[15] )
      Move(in := "Prior".DIFF_Prior, out1 => "BIASDIFF".DIFF)
   END_RUNG
   RUNG wire#powerrail
      I_Contact( "Params".stp_PARAMS[15] )
      Move(in := "StepVals".initDIFF, out1 => "BIASDIFF".DIFF)
   END_RUNG
   RUNG wire#powerrail
      Contact( "Params".stp_PARAMS[16] )
      Mul(in1 := "BIASDIFF".BIAS, in2 := 2.0, out => "BIASDIFF".DIFF)
   END_RUNG
   RUNG wire#powerrail
      Contact( "Params".stp_PARAMS[17] )
      Mul(in1 := -1.0, in2 := "BIASDIFF".DIFF, out => "BIASDIFF".DIFF)
   END_RUNG
   // the same network as SCL:
   IF "Params".stp_PARAMS[13] THEN "ANALOG_IO".remEfDrSP := "Prior".EfDr_Prior; END_IF;
   #_w1 := NOT "Params".stp_PARAMS[13];
   IF #_w1 AND "Params".stp_PARAMS[25] THEN "ANALOG_IO".remEfDrSP := "ref".EfDr_ref; END_IF;
   IF #_w1 AND NOT "Params".stp_PARAMS[25] THEN "ANALOG_IO".remEfDrSP := "StepVals".initEfDr; END_IF;
   IF "Params".stp_PARAMS[14] THEN "BIASDIFF".BIAS := "Prior".BIAS_Prior; END_IF;
   IF NOT "Params".stp_PARAMS[14] THEN "BIASDIFF".BIAS := "StepVals".initBIAS; END_IF;
   IF "Params".stp_PARAMS[24] THEN
       "StepVals".initBIAS := "ref".BIAS_ref;
       "BIASDIFF".BIAS := "StepVals".initBIAS;
   END_IF;
   IF "Params".stp_PARAMS[15] THEN "BIASDIFF".DIFF := "Prior".DIFF_Prior; END_IF;
   IF NOT "Params".stp_PARAMS[15] THEN "BIASDIFF".DIFF := "StepVals".initDIFF; END_IF;
   IF "Params".stp_PARAMS[16] THEN "BIASDIFF".DIFF := "BIASDIFF".BIAS * 2.0; END_IF;
   IF "Params".stp_PARAMS[17] THEN "BIASDIFF".DIFF := (-1.0) * "BIASDIFF".DIFF; END_IF;
END_REGION

REGION Network 6
   RUNG wire#powerrail
      "cam_zer_rdgs"()
   END_RUNG
   RUNG wire#powerrail
      Move(in := 0, out1 => "pulse".pulse_KV)
      Move(in := 0, out1 => "pulse".pulse_MA)
      Move(in := 0, out1 => "pulse".pulse_If)
   END_RUNG
   RUNG wire#powerrail
      Move(in := 0, out1 => "pulse".pulse_EfDr)
      Move(in := 0, out1 => "pulse".pulse_G1)
      Move(in := 0, out1 => "pulse".pulse_G2)
   END_RUNG
   // the same network as SCL:
   "cam_zer_rdgs"();
   "pulse".pulse_KV := 0;
   "pulse".pulse_MA := 0;
   "pulse".pulse_If := 0;
   "pulse".pulse_EfDr := 0;
   "pulse".pulse_G1 := 0;
   "pulse".pulse_G2 := 0;
END_REGION
END_FUNCTION_BLOCK

FUNCTION_BLOCK "Run_Sched"   // FB6, LAD
{ S7_Optimized_Access := 'TRUE' }
VERSION : 0.1
   VAR
      Step_Values_Instance : "Step_Values";
   END_VAR
   VAR RETAIN
      "step" : Int;
   END_VAR
   VAR
      stepdone : Bool;
      Run_Step_Instance : "Run_Step";
      retesttoend : Bool;
      tempsched_Instance : "tempsched";
   END_VAR
   VAR_TEMP   // added for the SCL form of the ladder/FBD networks
      _w1 : Bool;
   END_VAR
BEGIN

REGION Network 1: set current step to start step
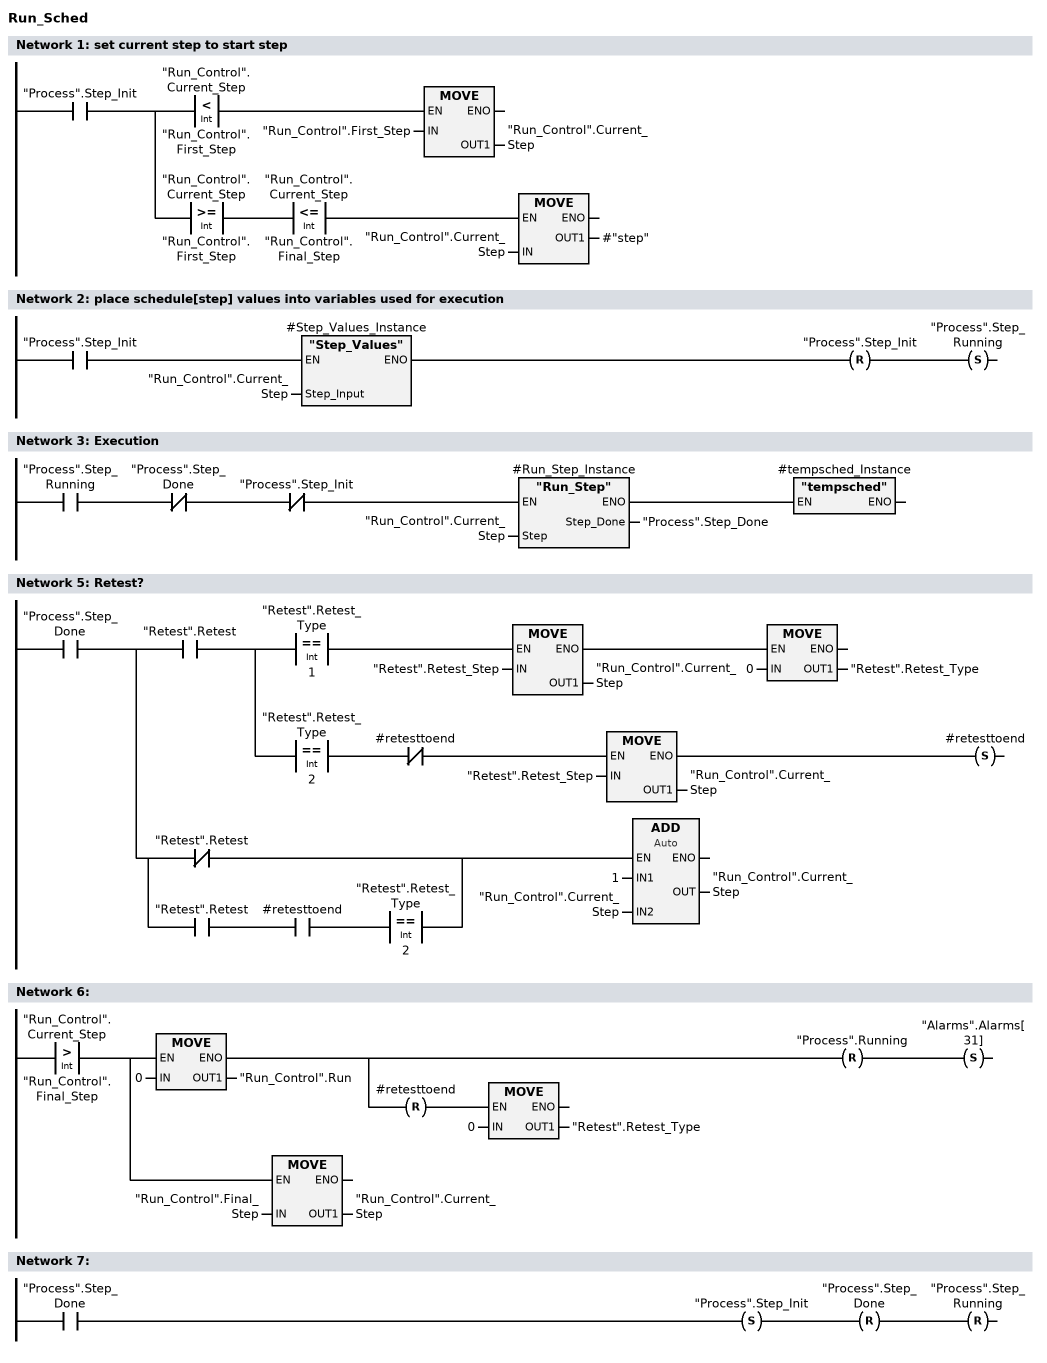
   RUNG wire#powerrail
      Contact( "Process".Step_Init )
      wire#w1
      { S7_Templates := "SrcType := Int" } LT_Contact(in1 := "Run_Control".Current_Step, in2 := "Run_Control".First_Step)
      Move(in := "Run_Control".First_Step, out1 => "Run_Control".Current_Step)
   END_RUNG
   RUNG wire#w1
      { S7_Templates := "SrcType := Int" } GE_Contact(in1 := "Run_Control".Current_Step, in2 := "Run_Control".First_Step)
      { S7_Templates := "SrcType := Int" } LE_Contact(in1 := "Run_Control".Current_Step, in2 := "Run_Control".Final_Step)
      Move(in := "Run_Control".Current_Step, out1 => #"step")
   END_RUNG
   // the same network as SCL:
   IF "Process".Step_Init AND ("Run_Control".Current_Step < "Run_Control".First_Step) THEN
       "Run_Control".Current_Step := "Run_Control".First_Step;
   END_IF;
   IF "Process".Step_Init AND ("Run_Control".Current_Step >= "Run_Control".First_Step) AND ("Run_Control".Current_Step <= "Run_Control".Final_Step) THEN
       #"step" := "Run_Control".Current_Step;
   END_IF;
END_REGION

REGION Network 2: place schedule[step] values into variables used for execution
   RUNG wire#powerrail
      Contact( "Process".Step_Init )
      #Step_Values_Instance(Step_Input := "Run_Control".Current_Step)
      R_Coil( "Process".Step_Init )
      S_Coil( "Process".Step_Running )
   END_RUNG
   // the same network as SCL:
   #Step_Values_Instance(EN := "Process".Step_Init, Step_Input := "Run_Control".Current_Step, ENO => #_w1);   // "Step_Values"
   IF #_w1 THEN
       "Process".Step_Init := FALSE;
       "Process".Step_Running := TRUE;
   END_IF;
END_REGION

REGION Network 3: Execution
   RUNG wire#powerrail
      Contact( "Process".Step_Running )
      I_Contact( "Process".Step_Done )
      I_Contact( "Process".Step_Init )
      #Run_Step_Instance("Step" := "Run_Control".Current_Step, Step_Done => "Process".Step_Done)
      #tempsched_Instance()
   END_RUNG
   // the same network as SCL:
   #Run_Step_Instance(EN := "Process".Step_Running AND NOT "Process".Step_Done AND NOT "Process".Step_Init,   // "Run_Step"
                      "Step" := "Run_Control".Current_Step,
                      Step_Done => "Process".Step_Done,
                      ENO => #_w1);
   IF #_w1 THEN
       #tempsched_Instance();   // "tempsched"
   END_IF;
END_REGION

REGION Network 4: TEST
END_REGION

REGION Network 5: Retest?
   RUNG wire#powerrail
      Contact( "Process".Step_Done )
      wire#w1
      Contact( "Retest".Retest )
      wire#w2
      { S7_Templates := "SrcType := Int" } EQ_Contact(in1 := "Retest".Retest_Type, in2 := 1)
      Move(in := "Retest".Retest_Step, out1 => "Run_Control".Current_Step)
      Move(in := 0, out1 => "Retest".Retest_Type)
   END_RUNG
   RUNG wire#w2
      { S7_Templates := "SrcType := Int" } EQ_Contact(in1 := "Retest".Retest_Type, in2 := 2)
      I_Contact( #retesttoend )
      Move(in := "Retest".Retest_Step, out1 => "Run_Control".Current_Step)
      S_Coil( #retesttoend )
   END_RUNG
   RUNG wire#w1
      I_Contact( "Retest".Retest )
      wire#w3
      Add(in1 := 1, in2 := "Run_Control".Current_Step, out => "Run_Control".Current_Step)
   END_RUNG
   RUNG wire#w1
      Contact( "Retest".Retest )
      Contact( #retesttoend )
      { S7_Templates := "SrcType := Int" } EQ_Contact(in1 := "Retest".Retest_Type, in2 := 2)
   END_RUNG wire#w3
   // the same network as SCL:
   #_w1 := "Process".Step_Done AND "Retest".Retest;
   IF #_w1 AND ("Retest".Retest_Type = 1) THEN
       "Run_Control".Current_Step := "Retest".Retest_Step;
       "Retest".Retest_Type := 0;
   END_IF;
   IF #_w1 AND ("Retest".Retest_Type = 2) AND NOT #retesttoend THEN
       "Run_Control".Current_Step := "Retest".Retest_Step;
       #retesttoend := TRUE;
   END_IF;
   IF "Process".Step_Done AND (NOT "Retest".Retest OR ("Retest".Retest AND #retesttoend AND ("Retest".Retest_Type = 2))) THEN
       "Run_Control".Current_Step := 1 + "Run_Control".Current_Step;
   END_IF;
END_REGION

REGION Network 6
   RUNG wire#powerrail
      { S7_Templates := "SrcType := Int" } GT_Contact(in1 := "Run_Control".Current_Step, in2 := "Run_Control".Final_Step)
      wire#w1
      Move(in := 0, out1 => "Run_Control".Run)
      wire#w2
      R_Coil( "Process".Running )
      S_Coil( "Alarms".Alarms[31] )
   END_RUNG
   RUNG wire#w2
      R_Coil( #retesttoend )
      Move(in := 0, out1 => "Retest".Retest_Type)
   END_RUNG
   RUNG wire#w1
      Move(in := "Run_Control".Final_Step, out1 => "Run_Control".Current_Step)
   END_RUNG
   // the same network as SCL:
   IF "Run_Control".Current_Step > "Run_Control".Final_Step THEN
       "Run_Control".Run := 0;
       "Process".Running := FALSE;
       "Alarms".Alarms[31] := TRUE;
       #retesttoend := FALSE;
       "Retest".Retest_Type := 0;
       "Run_Control".Current_Step := "Run_Control".Final_Step;
   END_IF;
END_REGION

REGION Network 7
   RUNG wire#powerrail
      Contact( "Process".Step_Done )
      S_Coil( "Process".Step_Init )
      R_Coil( "Process".Step_Done )
      R_Coil( "Process".Step_Running )
   END_RUNG
   // the same network as SCL:
   IF "Process".Step_Done THEN "Process".Step_Init := TRUE; END_IF;
   #_w1 := "Process".Step_Done;
   IF #_w1 THEN
       "Process".Step_Done := FALSE;
       "Process".Step_Running := FALSE;
   END_IF;
END_REGION
END_FUNCTION_BLOCK

FUNCTION_BLOCK "ALARMS_CHECK"   // FB9, LAD
{ S7_Optimized_Access := 'TRUE' }
VERSION : 0.1
   VAR_TEMP
      alarms_inverted : Array[0..31] of Bool;
      Alarmcheck : Bool;
      c : Int;
      c2 : Int;
      Proccheck : Bool;
   END_VAR
BEGIN

REGION Network 2 (SCL)
   FOR #c := 0 TO 31 DO
       #Alarmcheck := #Alarmcheck OR "Alarms".Alarms[#c];
   END_FOR;
END_REGION

REGION Network 3
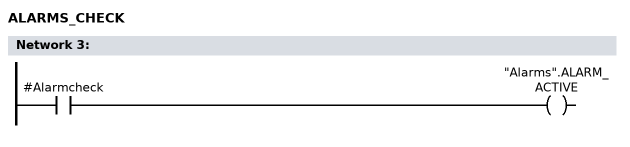
   RUNG wire#powerrail
      Contact( #Alarmcheck )
      Coil( "Alarms".ALARM_ACTIVE )
   END_RUNG
   // the same network as SCL:
   "Alarms".ALARM_ACTIVE := #Alarmcheck;
END_REGION

REGION Network 4 (SCL)
   IF "Alarms".Alarm_Clear THEN
       FOR #c2 := 0 TO 31 DO
           "Alarms".Alarms[#c2] := FALSE;
       END_FOR;
       "Alarms".Alarm_Clear := FALSE;
   END_IF;
END_REGION
END_FUNCTION_BLOCK

FUNCTION_BLOCK "Reset"   // FB10, LAD
{ S7_Optimized_Access := 'TRUE' }
VERSION : 0.1
   VAR_TEMP
      c : Int;
   END_VAR
BEGIN

REGION Network 2 (SCL)
   "Run_Control".Run := 0;
   "Run_Control".First_Step := 0;
   "Run_Control".Current_Step := 0;
   "Run_Control".Final_Step := 0;
   "Process".Run_Init := TRUE;
   "Process".Step_Init := TRUE;
   "Process".Running := FALSE;
   "Process".Step_Running := FALSE;
   "Process".Step_Done := FALSE;
   "Process".Schedule_Done := FALSE;
   "Process".Retest_Done := FALSE;
   "Process".Results_Ready := FALSE;

   "StepVals".COOLtime := 0;
   "StepVals".dataitem := 0;
   "StepVals".EXPtime := 0;
   "StepVals".initBIAS := 0;
   "StepVals".initDIFF := 0;
   "StepVals".initEfDr := 0;
   "StepVals".KV := 0;
   "StepVals".LIM1 := 0;
   "StepVals".LIM2 := 0;
   "StepVals".LIM3 := 0;
   "StepVals".LIM4 := 0;
   "StepVals".MAIf := 0;
   "StepVals".max := 0;
   "StepVals".maxGx := 0;
   "StepVals".maxTries := 0;
   "StepVals".min := 0;
   "StepVals".PARAMS := 0;
   "StepVals".scansMode := 0;
   "StepVals".TEST := 0;

   "ANALOG_IO".G1V_SP := 0;
   "ANALOG_IO".G2V_SP := 0;
   "ANALOG_IO".remEfDrSP := 0;
   "ANALOG_IO".remKVSP := 0;
   "ANALOG_IO".remMASP := 0;

   "Alarms".Alarms[31] := FALSE;
END_REGION
END_FUNCTION_BLOCK

FUNCTION_BLOCK "Heat_Int"   // FB11, LAD
{ S7_Optimized_Access := 'TRUE' }
VERSION : 0.1
   VAR
      Watts : Real;
      Heat_Int_t : Time := T#10000ms;
      Heat_Int_Tmr : TON_TIME;
      Heat_Storage : Real;
   END_VAR
   VAR_TEMP
      heat_int_timer_temp : Real;
   END_VAR
BEGIN

REGION Network 1 (SCL)
   #Heat_Int_Tmr(IN:=TRUE,
                 PT:=#Heat_Int_t);

   IF ("ANALOG_IO".remKVrdg > 3.0) AND ("ANALOG_IO".remMArdg > 3.0) THEN
       #Watts := "ANALOG_IO".remKVrdg * "ANALOG_IO".remMArdg;
   ELSE
       #Watts := 0;
   END_IF;
   #heat_int_timer_temp := INT_TO_REAL(TIME_TO_INT(#Heat_Int_Tmr.ET));
   "System".Temp_rdg := "System".Temp_rdg + (#Watts * "Tube".AP / 100.0 - "Tube".RTC * (10**-011) *("System".Temp_rdg + 273.0)**4) * ("Tube".T100 - "Tube".T0) / "Tube".HS / 1000 * #heat_int_timer_temp / 1000;

   IF "System".Temp_rdg < "Tube".T0 THEN
       "System".Temp_rdg := 0;
   END_IF;
   #Heat_Storage := ("System".Temp_rdg - "Tube".T0) / ("Tube".T100 - "Tube".T0) * 100;
   RESET_TIMER(#Heat_Int_Tmr);

   IF "System".Temp_set > -0.1 THEN
       "System".Temp_rdg := "System".Temp_set;
       "System".Temp_set := -0.1;
   END_IF;
   IF "System".Temp_rdg > "Limits".LIMITS[13] THEN
       "Alarms".Alarms[11] := TRUE;
       "Run_Control".Reset := 1;   //Turn on Reset
       "System".Sleep := TRUE;     //Turn on Sleep
       //Set Status: "TEMP>LIMITS[13] ABORT"
   END_IF;
END_REGION
END_FUNCTION_BLOCK

// folder: Sub Routines

FUNCTION_BLOCK "Moving_Avg"   // FB4, LAD
{ S7_Optimized_Access := 'TRUE' }
VERSION : 0.1
   VAR_INPUT
      NewInput : DInt;
   END_VAR
   VAR_OUTPUT
      AvgOutput : DInt;
   END_VAR
   VAR RETAIN
      OldVal : DInt;
   END_VAR
   VAR_TEMP
      array_idx : Int;
      avg : DInt;
   END_VAR
   VAR CONSTANT
      Window_size : Int := 8;
   END_VAR
BEGIN

REGION Network 1 (SCL)
   IF #OldVal < (0.5*#NewInput)  THEN
       #AvgOutput := #NewInput;
   ELSE
       #AvgOutput := (#NewInput + #OldVal) / 2;
   END_IF;

   #OldVal := #AvgOutput;
END_REGION
END_FUNCTION_BLOCK

FUNCTION_BLOCK "Run_Step"   // FB7, LAD
{ S7_Optimized_Access := 'TRUE' }
VERSION : 0.1
   VAR_INPUT
      "Step" : Int;
   END_VAR
   VAR_OUTPUT
      Step_Done : Bool;
   END_VAR
   VAR
      substep : Int;
      ProcNOKtmr : TON_TIME;
      XPOSE_TMR1 : TON_TIME;
   END_VAR
   VAR_TEMP
      compile : Bool;
   END_VAR
   VAR_TEMP   // added for the SCL form of the ladder/FBD networks
      _w1 : Bool;
      _w2 : Bool;
   END_VAR
BEGIN

REGION Network 1: Process Check
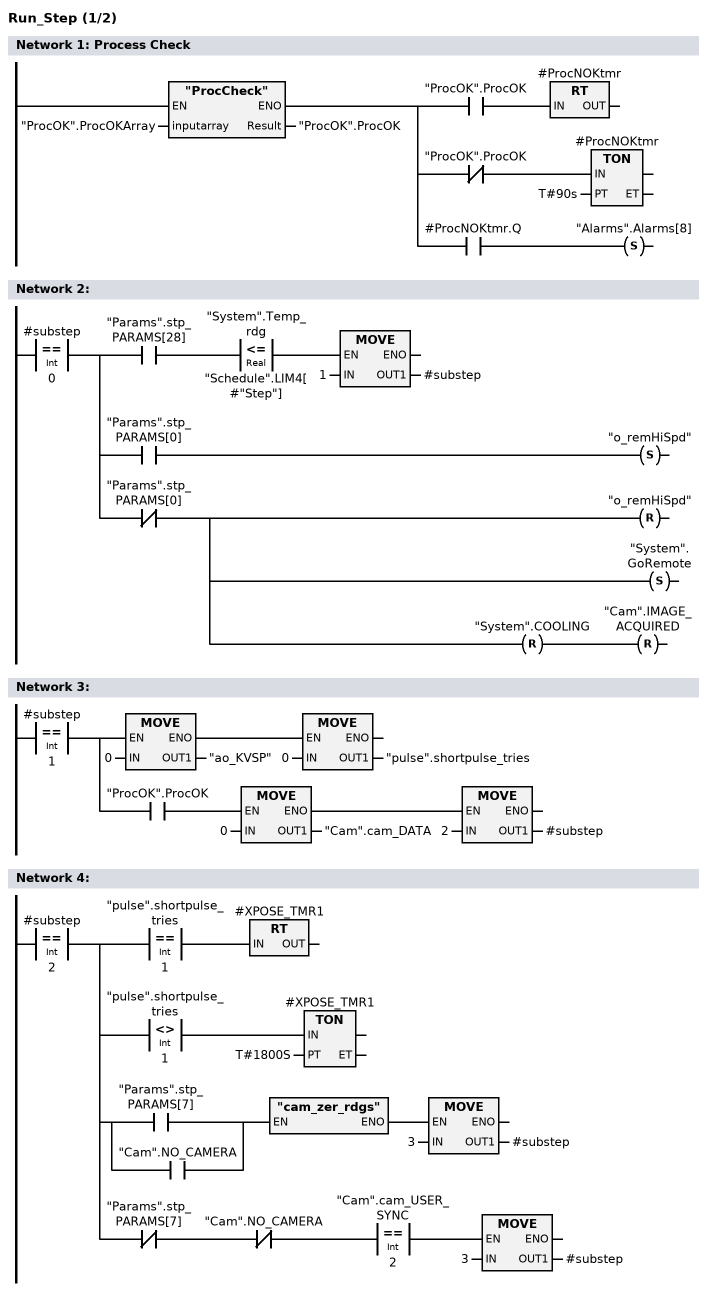
   "ProcCheck"(inputarray := "ProcOK".ProcOKArray, Result => "ProcOK".ProcOK, ENO => #_w1);
   IF #_w1 AND "ProcOK".ProcOK THEN RESET_TIMER(#ProcNOKtmr); END_IF;
   #ProcNOKtmr(IN := #_w1 AND NOT "ProcOK".ProcOK, PT := T#90s);   // TON
   IF #_w1 AND #ProcNOKtmr.Q THEN "Alarms".Alarms[8] := TRUE; END_IF;
END_REGION

REGION Network 2
   RUNG wire#powerrail
      { S7_Templates := "SrcType := Int" } EQ_Contact(in1 := #substep, in2 := 0)
      wire#w1
      Contact( "Params".stp_PARAMS[28] )
      { S7_Templates := "SrcType := Real" } LE_Contact(in1 := "System".Temp_rdg, in2 := "Schedule".LIM4[#"Step"])
      Move(in := 1, out1 => #substep)
   END_RUNG
   RUNG wire#w1
      Contact( "Params".stp_PARAMS[0] )
      S_Coil( "o_remHiSpd" )
   END_RUNG
   RUNG wire#w1
      I_Contact( "Params".stp_PARAMS[0] )
      wire#w2
      R_Coil( "o_remHiSpd" )
   END_RUNG
   RUNG wire#w2
      S_Coil( "System".GoRemote )
   END_RUNG
   RUNG wire#w2
      R_Coil( "System".COOLING )
      R_Coil( "Cam".IMAGE_ACQUIRED )
   END_RUNG
   // the same network as SCL:
   #_w1 := #substep = 0;
   IF #_w1 AND "Params".stp_PARAMS[28] AND ("System".Temp_rdg <= "Schedule".LIM4[#"Step"]) THEN
       #substep := 1;
   END_IF;
   IF #_w1 AND "Params".stp_PARAMS[0] THEN "o_remHiSpd" := TRUE; END_IF;
   IF #_w1 AND NOT "Params".stp_PARAMS[0] THEN
       "o_remHiSpd" := FALSE;
       "System".GoRemote := TRUE;
       "System".COOLING := FALSE;
       "Cam".IMAGE_ACQUIRED := FALSE;
   END_IF;
END_REGION

REGION Network 3
   RUNG wire#powerrail
      { S7_Templates := "SrcType := Int" } EQ_Contact(in1 := #substep, in2 := 1)
      wire#w1
      Move(in := 0, out1 => "ao_KVSP")
      Move(in := 0, out1 => "pulse".shortpulse_tries)
   END_RUNG
   RUNG wire#w1
      Contact( "ProcOK".ProcOK )
      Move(in := 0, out1 => "Cam".cam_DATA)
      Move(in := 2, out1 => #substep)
   END_RUNG
   // the same network as SCL:
   #_w1 := #substep = 1;
   IF #_w1 THEN
       "ao_KVSP" := 0;
       "pulse".shortpulse_tries := 0;
   END_IF;
   IF #_w1 AND "ProcOK".ProcOK THEN
       "Cam".cam_DATA := 0;
       #substep := 2;
   END_IF;
END_REGION

REGION Network 4
   #_w1 := #substep = 2;
   IF #_w1 AND ("pulse".shortpulse_tries = 1) THEN RESET_TIMER(#XPOSE_TMR1); END_IF;
   #XPOSE_TMR1(IN := #_w1 AND ("pulse".shortpulse_tries <> 1), PT := T#1800S);   // TON
   "cam_zer_rdgs"(EN := #_w1 AND ("Params".stp_PARAMS[7] OR "Cam".NO_CAMERA), ENO => #_w2);
   IF #_w2 THEN #substep := 3; END_IF;
   IF #_w1 AND NOT "Params".stp_PARAMS[7] AND NOT "Cam".NO_CAMERA AND ("Cam".cam_USER_SYNC = 2) THEN
       #substep := 3;
   END_IF;
END_REGION

REGION Network 5: pulse exposure
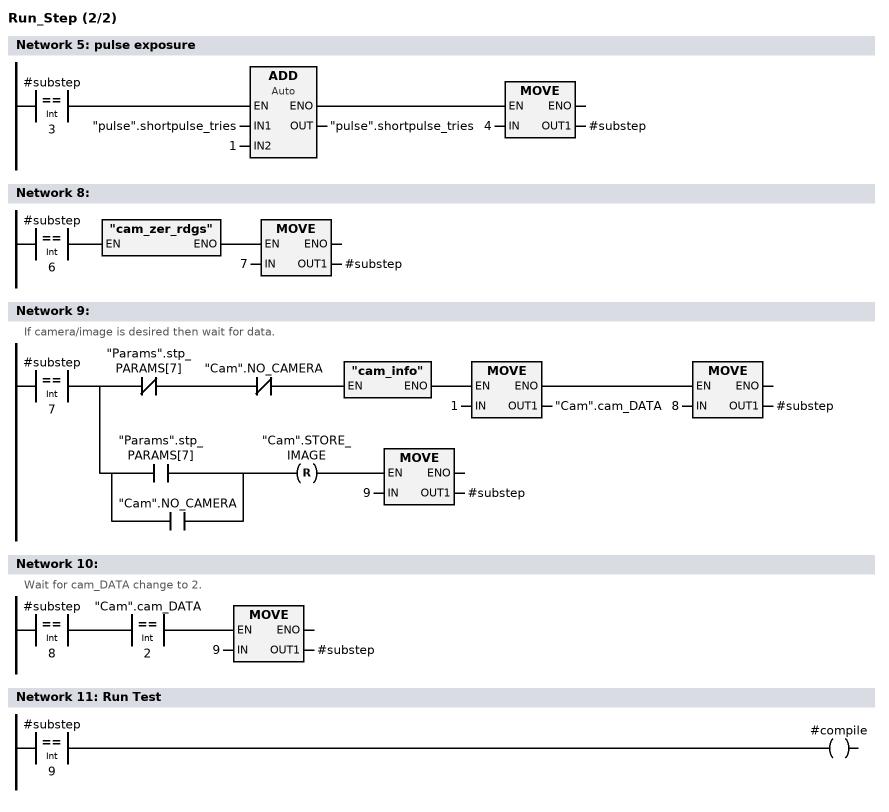
   RUNG wire#powerrail
      { S7_Templates := "SrcType := Int" } EQ_Contact(in1 := #substep, in2 := 3)
      Add(in1 := "pulse".shortpulse_tries, in2 := 1, out => "pulse".shortpulse_tries)
      Move(in := 4, out1 => #substep)
   END_RUNG
   // the same network as SCL:
   IF #substep = 3 THEN
       "pulse".shortpulse_tries := "pulse".shortpulse_tries + 1;
       #substep := 4;
   END_IF;
END_REGION

REGION Network 6 (SCL): Check temperature limits
   IF #substep = 4 THEN
       IF ("Params".stp_PARAMS[1] AND ("System".Temp_rdg > "Limits".LIMITS[32])) THEN
           "StepVals".EXPtime := 0.0;
           "ao_KVSP" := 0;
       END_IF;
       IF ("Params".stp_PARAMS[1] AND ("System".Temp_rdg > "Limits".LIMITS[32])) THEN
           "ao_KVSP" := 0;
       ELSE
           #substep := 5;
       END_IF;
   END_IF;
END_REGION

REGION Network 7 (SCL)
   IF #substep = 5 THEN
       IF "StepVals".EXPtime >= "pulse".pulsePeriod THEN
           IF "pulse".XPOSE_SEC <= "StepVals".EXPtime THEN
               "pulse".shortpulse_tries := 2;
               IF "Params".stp_PARAMS[1] AND ("System".Temp_rdg > "Limits".LIMITS[32]) THEN
                   "StepVals".EXPtime := 0;
                   "ao_KVSP" := 0;
                   #substep := 6;
               ELSE
                   "Cam".cam_DATA := 0;
                   #substep := 2;
               END_IF;
           ELSE
               #substep := 6;
           END_IF;
       ELSE
           IF "System".Exp_MA_If_OK = FALSE THEN
               IF "pulse".shortpulse_tries > "Limits".LIMITS[9] THEN
                   //Jump to later step.
                   RESET_TIMER(#XPOSE_TMR1);
                   "Alarms".Alarms[7] := TRUE;
                   "Run_Control".Reset := 1;
                   ;
               ELSE
                   #substep := 2;
               END_IF;
           ELSE
               #substep := 6;
           END_IF;
       END_IF;
   END_IF;
END_REGION

REGION Network 8
   RUNG wire#powerrail
      { S7_Templates := "SrcType := Int" } EQ_Contact(in1 := #substep, in2 := 6)
      "cam_zer_rdgs"()
      Move(in := 7, out1 => #substep)
   END_RUNG
   // the same network as SCL:
   "cam_zer_rdgs"(EN := #substep = 6, ENO => #_w1);
   IF #_w1 THEN #substep := 7; END_IF;
END_REGION

REGION Network 9
   // If camera/image is desired then wait for data.
   RUNG wire#powerrail
      { S7_Templates := "SrcType := Int" } EQ_Contact(in1 := #substep, in2 := 7)
      wire#w1
      I_Contact( "Params".stp_PARAMS[7] )
      I_Contact( "Cam".NO_CAMERA )
      "cam_info"()
      Move(in := 1, out1 => "Cam".cam_DATA)
      Move(in := 8, out1 => #substep)
   END_RUNG
   RUNG wire#w1
      Contact( "Params".stp_PARAMS[7] )
      wire#w2
      R_Coil( "Cam".STORE_IMAGE )
      Move(in := 9, out1 => #substep)
   END_RUNG
   RUNG wire#w1
      Contact( "Cam".NO_CAMERA )
   END_RUNG wire#w2
   // the same network as SCL:
   #_w1 := #substep = 7;
   "cam_info"(EN := #_w1 AND NOT "Params".stp_PARAMS[7] AND NOT "Cam".NO_CAMERA, ENO => #_w2);
   IF #_w2 THEN
       "Cam".cam_DATA := 1;
       #substep := 8;
   END_IF;
   IF #_w1 AND ("Params".stp_PARAMS[7] OR "Cam".NO_CAMERA) THEN
       "Cam".STORE_IMAGE := FALSE;
       #substep := 9;
   END_IF;
END_REGION

REGION Network 10
   // Wait for cam_DATA change to 2.
   RUNG wire#powerrail
      { S7_Templates := "SrcType := Int" } EQ_Contact(in1 := #substep, in2 := 8)
      { S7_Templates := "SrcType := Int" } EQ_Contact(in1 := "Cam".cam_DATA, in2 := 2)
      Move(in := 9, out1 => #substep)
   END_RUNG
   // the same network as SCL:
   IF (#substep = 8) AND ("Cam".cam_DATA = 2) THEN #substep := 9; END_IF;
END_REGION

REGION Network 11: Run Test
   RUNG wire#powerrail
      { S7_Templates := "SrcType := Int" } EQ_Contact(in1 := #substep, in2 := 9)
      Coil( #compile )
   END_RUNG
   // the same network as SCL:
   #compile := #substep = 9;
END_REGION
END_FUNCTION_BLOCK

FUNCTION_BLOCK "TEST"   // FB8, LAD
{ S7_Optimized_Access := 'TRUE' }
VERSION : 0.1
   VAR_TEMP
      substep : Int;
      temp : Bool;
   END_VAR
   VAR_TEMP   // added for the SCL form of the ladder/FBD networks
      _w1 : Bool;
      _w2 : Bool;
      _w3 : Bool;
      _w4 : Bool;
      _w5 : Bool;
      _w6 : Bool;
      _w7 : Bool;
   END_VAR
BEGIN

REGION Network 1
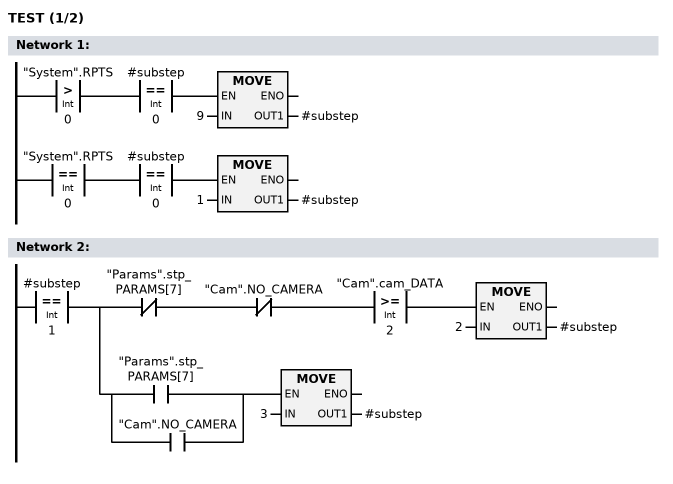
   RUNG wire#powerrail
      { S7_Templates := "SrcType := Int" } GT_Contact(in1 := "System".RPTS, in2 := 0)
      { S7_Templates := "SrcType := Int" } EQ_Contact(in1 := #substep, in2 := 0)
      Move(in := 9, out1 => #substep)
   END_RUNG
   RUNG wire#powerrail
      { S7_Templates := "SrcType := Int" } EQ_Contact(in1 := "System".RPTS, in2 := 0)
      { S7_Templates := "SrcType := Int" } EQ_Contact(in1 := #substep, in2 := 0)
      Move(in := 1, out1 => #substep)
   END_RUNG
   // the same network as SCL:
   IF ("System".RPTS > 0) AND (#substep = 0) THEN #substep := 9; END_IF;
   IF ("System".RPTS = 0) AND (#substep = 0) THEN #substep := 1; END_IF;
END_REGION

REGION Network 2
   RUNG wire#powerrail
      { S7_Templates := "SrcType := Int" } EQ_Contact(in1 := #substep, in2 := 1)
      wire#w1
      I_Contact( "Params".stp_PARAMS[7] )
      I_Contact( "Cam".NO_CAMERA )
      { S7_Templates := "SrcType := Int" } GE_Contact(in1 := "Cam".cam_DATA, in2 := 2)
      Move(in := 2, out1 => #substep)
   END_RUNG
   RUNG wire#w1
      Contact( "Params".stp_PARAMS[7] )
      wire#w2
      Move(in := 3, out1 => #substep)
   END_RUNG
   RUNG wire#w1
      Contact( "Cam".NO_CAMERA )
   END_RUNG wire#w2
   // the same network as SCL:
   #_w1 := #substep = 1;
   IF #_w1 AND NOT "Params".stp_PARAMS[7] AND NOT "Cam".NO_CAMERA AND ("Cam".cam_DATA >= 2) THEN
       #substep := 2;
   END_IF;
   IF #_w1 AND ("Params".stp_PARAMS[7] OR "Cam".NO_CAMERA) THEN #substep := 3; END_IF;
END_REGION

REGION Network 3 (SCL)
   IF #substep = 2 THEN
       IF "Params".stp_TEST[0] THEN
           "ref".BIAS_ref := "BIASDIFF".BIAS;
       END_IF;
       IF "Params".stp_TEST[1] THEN
           "Cam".cam_Xref := "Cam".cam_Xpos - "Limits".LIMITS[23];
           "Cam".cam_Zref := "Cam".cam_Zpos - "Limits".LIMITS[24];
           "Cam".cam_Yref := "Cam".cam_Ypos - "Limits".LIMITS[25];
       END_IF;
       IF "Params".stp_TEST[2] THEN
           "Cam".X_defl := ROUND(("Cam".cam_Xpos - "Limits".LIMITS[23] - "Cam".cam_Xref) * 1000) / 1000;
           "MIN_MAX"(TESTVAL := "Cam".X_defl,
                     Pass_Fail => "Results".Pass_Fail);
           "Results".testVAL := "Cam".X_defl;
       END_IF;
       IF "Params".stp_TEST[3] THEN
           "MIN_MAX"(TESTVAL := "Cam".cam_WIDTH,
                     Pass_Fail => "Results".Pass_Fail);
           "Results".testVAL := ROUND(1000 * "Cam".cam_WIDTH) / 1000;
       END_IF;
       IF "Params".stp_TEST[4] THEN
           "MIN_MAX"(TESTVAL := "Cam".cam_LENGTH,
                     Pass_Fail => "Results".Pass_Fail);
           "Results".testVAL := ROUND(1000 * "Cam".cam_LENGTH) / 1000;
       END_IF;
       #substep := 3;
   END_IF;
END_REGION

REGION Network 4
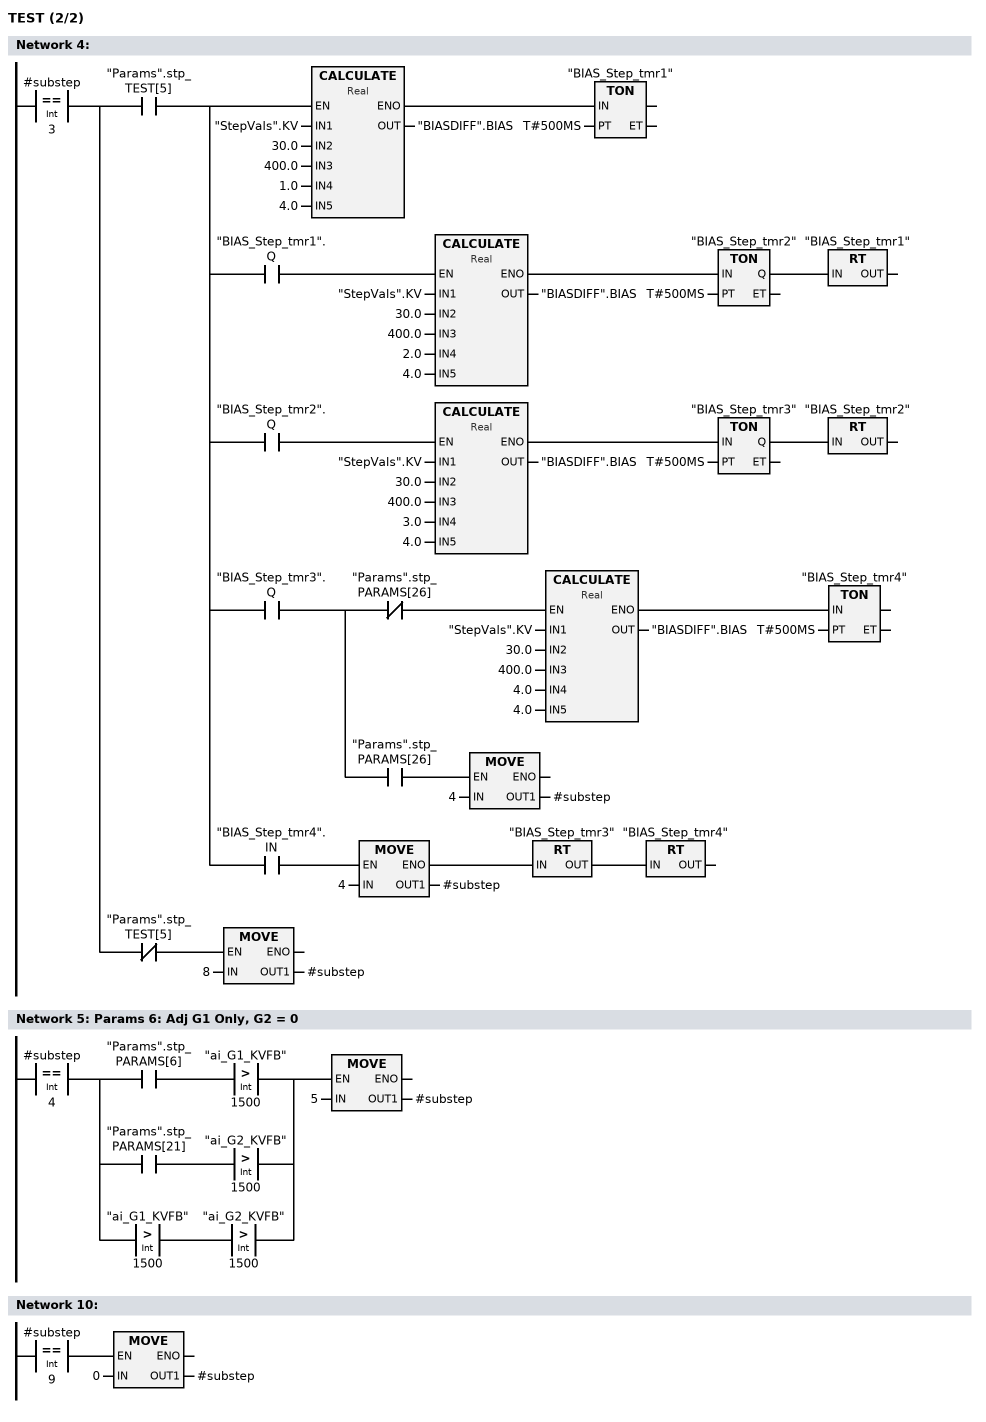
   #_w1 := #substep = 3;
   #_w2 := #_w1 AND "Params".stp_TEST[5];
   IF #_w2 THEN "BIASDIFF".BIAS := ("StepVals".KV*30.0 - 400.0) * 1.0 / 4.0; END_IF;
   "BIAS_Step_tmr1".TON(IN := #_w2, PT := T#500MS);
   #_w3 := #_w2 AND "BIAS_Step_tmr1".Q;
   IF #_w3 THEN "BIASDIFF".BIAS := ("StepVals".KV*30.0 - 400.0) * 2.0 / 4.0; END_IF;
   "BIAS_Step_tmr2".TON(IN := #_w3, PT := T#500MS);
   IF "BIAS_Step_tmr2".Q THEN RESET_TIMER("BIAS_Step_tmr1"); END_IF;
   #_w4 := #_w2 AND "BIAS_Step_tmr2".Q;
   IF #_w4 THEN "BIASDIFF".BIAS := ("StepVals".KV*30.0 - 400.0) * 3.0 / 4.0; END_IF;
   "BIAS_Step_tmr3".TON(IN := #_w4, PT := T#500MS);
   IF "BIAS_Step_tmr3".Q THEN RESET_TIMER("BIAS_Step_tmr2"); END_IF;
   #_w5 := #_w2 AND "BIAS_Step_tmr3".Q;
   #_w6 := #_w5 AND NOT "Params".stp_PARAMS[26];
   IF #_w6 THEN "BIASDIFF".BIAS := ("StepVals".KV*30.0 - 400.0) * 4.0 / 4.0; END_IF;
   "BIAS_Step_tmr4".TON(IN := #_w6, PT := T#500MS);
   IF #_w5 AND "Params".stp_PARAMS[26] THEN #substep := 4; END_IF;
   #_w7 := #_w2 AND "BIAS_Step_tmr4".IN;
   IF #_w7 THEN
       #substep := 4;
       RESET_TIMER("BIAS_Step_tmr3");
       RESET_TIMER("BIAS_Step_tmr4");
   END_IF;
   IF #_w1 AND NOT "Params".stp_TEST[5] THEN #substep := 8; END_IF;
END_REGION

REGION Network 5: Params 6: Adj G1 Only, G2 = 0
   RUNG wire#powerrail
      { S7_Templates := "SrcType := Int" } EQ_Contact(in1 := #substep, in2 := 4)
      wire#w1
      Contact( "Params".stp_PARAMS[6] )
      { S7_Templates := "SrcType := Int" } GT_Contact(in1 := "ai_G1_KVFB", in2 := 1500)
      wire#w2
      Move(in := 5, out1 => #substep)
   END_RUNG
   RUNG wire#w1
      Contact( "Params".stp_PARAMS[21] )
      { S7_Templates := "SrcType := Int" } GT_Contact(in1 := "ai_G2_KVFB", in2 := 1500)
   END_RUNG wire#w2
   RUNG wire#w1
      { S7_Templates := "SrcType := Int" } GT_Contact(in1 := "ai_G1_KVFB", in2 := 1500)
      { S7_Templates := "SrcType := Int" } GT_Contact(in1 := "ai_G2_KVFB", in2 := 1500)
   END_RUNG wire#w2
   // the same network as SCL:
   IF (#substep = 4) AND (("Params".stp_PARAMS[6] AND ("ai_G1_KVFB" > 1500)) OR ("Params".stp_PARAMS[21] AND ("ai_G2_KVFB" > 1500)) OR (("ai_G1_KVFB" > 1500) AND ("ai_G2_KVFB" > 1500))) THEN
       #substep := 5;
   END_IF;
END_REGION

REGION Network 6 (SCL)
   IF #substep = 5 THEN
       "ao_KVSP" := REAL_TO_INT("StepVals".KV);
       "Cutoff".cutoff_avg_MA := TRUE;
       #substep := 6;
   END_IF;
END_REGION

REGION Network 7 (SCL)
   IF #substep = 6 THEN
       IF "Misc".rem_MA_rdg_avg >"StepVals".LIM3 THEN
           "BIASDIFF".delta_BIAS := ("Misc".rem_MA_rdg_avg - 0.3) * "Limits".LIMITS[20];
           "CLAMP_FLOAT"(in:="BIASDIFF".delta_BIAS,
                         min:=5,
                         max:=20,
                         out=>"BIASDIFF".delta_BIAS);
           "BIASDIFF".BIAS := "BIASDIFF".BIAS + "BIASDIFF".delta_BIAS;
           "Gx".Gx_LIMIT := "StepVals".maxGx;
           "CLAMP_FLOAT"(in:="BIASDIFF".BIAS,
                         min:=0,
                         max:="Gx".Gx_LIMIT,
                         out=>"BIASDIFF".BIAS);
           IF "Params".stp_PARAMS[6] THEN
               "Cutoff".cutoff_BIAS := ROUND("ai_G1_KVFB");
           ELSE
               IF "Params".stp_PARAMS[21] THEN
                   "Cutoff".cutoff_BIAS := ROUND("ai_G2_KVFB");
               ELSE
                   "Cutoff".cutoff_BIAS := ROUND("ai_G1_KVFB" / 2 + "ai_G2_KVFB" / 2);
               END_IF;
           END_IF;
       ELSE
           #substep := 7;
       END_IF;
   END_IF;
END_REGION

REGION Network 8 (SCL)
   IF #substep = 7 THEN
       "MIN_MAX"(TESTVAL:="Cutoff".cutoff_BIAS,
                 Pass_Fail=>"Results".Pass_Fail);
       "Results".testVAL := "Cutoff".cutoff_BIAS;
       "BIASDIFF".BIAS := 0;
       "Cutoff".cutoff_avg_MA := FALSE;
       "pulse".pulse_G1 := "ai_G1_KVFB";
       "pulse".pulse_G2 := "ai_G2_KVFB";
       #substep := 8;
   END_IF;
END_REGION

REGION Network 9 (SCL)
   IF #substep = 8 THEN
       IF "Params".stp_TEST[6] THEN
           "ref".EfDr_ref := "Remote".remEfDr_SP;
       END_IF;
       IF "Params".stp_TEST[7] AND "Cam".cam_WIDTH < "StepVals".LIM3 THEN
           "Results".Pass_Fail := -1;
       END_IF;
       #substep := 9;
   END_IF;
END_REGION

REGION Network 10
   RUNG wire#powerrail
      { S7_Templates := "SrcType := Int" } EQ_Contact(in1 := #substep, in2 := 9)
      Move(in := 0, out1 => #substep)
   END_RUNG
   // the same network as SCL:
   IF #substep = 9 THEN #substep := 0; END_IF;
END_REGION
END_FUNCTION_BLOCK

FUNCTION_BLOCK "Retests"   // FB12, LAD
{ S7_Optimized_Access := 'TRUE' }
VERSION : 0.1
BEGIN

REGION Network 1
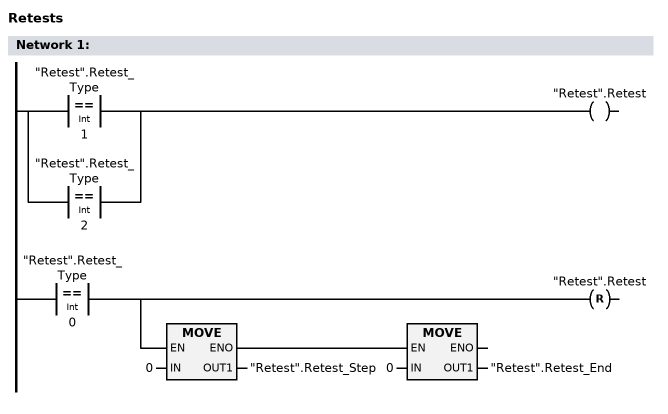
   RUNG wire#powerrail
      { S7_Templates := "SrcType := Int" } EQ_Contact(in1 := "Retest".Retest_Type, in2 := 1)
      wire#w1
      Coil( "Retest".Retest )
   END_RUNG
   RUNG wire#powerrail
      { S7_Templates := "SrcType := Int" } EQ_Contact(in1 := "Retest".Retest_Type, in2 := 2)
   END_RUNG wire#w1
   RUNG wire#powerrail
      { S7_Templates := "SrcType := Int" } EQ_Contact(in1 := "Retest".Retest_Type, in2 := 0)
      wire#w2
      R_Coil( "Retest".Retest )
   END_RUNG
   RUNG wire#w2
      Move(in := 0, out1 => "Retest".Retest_Step)
      Move(in := 0, out1 => "Retest".Retest_End)
   END_RUNG
   // the same network as SCL:
   "Retest".Retest := ("Retest".Retest_Type = 1) OR ("Retest".Retest_Type = 2);
   IF "Retest".Retest_Type = 0 THEN
       "Retest".Retest := FALSE;
       "Retest".Retest_Step := 0;
       "Retest".Retest_End := 0;
   END_IF;
END_REGION
END_FUNCTION_BLOCK

FUNCTION_BLOCK "tempsched"   // FB13, LAD
{ S7_Optimized_Access := 'TRUE' }
VERSION : 0.1
   VAR
      neg : Int := 1;
      IEC_Timer_0_Instance : TON_TIME;
   END_VAR
BEGIN

REGION Network 2 (SCL)

   #IEC_Timer_0_Instance(IN:=TRUE,
                         PT:=T#2s);
   "Process".Results_Ready := TRUE;
   IF #IEC_Timer_0_Instance.Q THEN
       "Results".dataitem := "StepVals".dataitem;
       "Results".EfDr := "StepVals".initEfDr;
       "Results".G1V := "Run_Control"."Current_Step";
       "Results".G2V := "Run_Control"."Current_Step" * -1;
       "Results"."If" := "StepVals".MAIf;
       "Results".KV := "StepVals".KV;
       "Results".Length := 0.64;
       "Results".MA := "StepVals".MAIf;
       "Results".Mag := "Run_Control"."Current_Step";
       "Results".max := "StepVals".max;
       "Results".min := "StepVals".min;
       "Results".OBpk := "Run_Control"."Current_Step";
       IF "Run_Control"."Current_Step" < 1 THEN
           "Results".Pass_Fail := 1;

       ELSE
           "Results".Pass_Fail := #neg;
       END_IF;

       "Results".pk := "Run_Control"."Current_Step";
       "Results".scansmode := "StepVals".scansMode;
       "Results".Temp := 100 + "Run_Control"."Current_Step";
       "Results".testVAL := "Run_Control"."Current_Step";
       "Results".tries := "StepVals".maxTries;
       "Results".Width := "Run_Control"."Current_Step";
       "Results".Xdefl := 1 + "Run_Control"."Current_Step";
       "Results".Xpos := "Run_Control"."Current_Step";
       "Results".Zdefl := 2 + "Run_Control"."Current_Step";
       "Results".Zpos := "Run_Control"."Current_Step";
       "Results".Ydefl := 3 + "Run_Control"."Current_Step";
       "Results".Ypos := "Run_Control"."Current_Step";
       "Process".Results_Ready := FALSE;
       "Process".Step_Done := TRUE;
       RESET_TIMER(#IEC_Timer_0_Instance);
       #IEC_Timer_0_Instance.IN := FALSE;
   END_IF;

   #neg := -1 * #neg;
END_REGION
END_FUNCTION_BLOCK

FUNCTION "CLAMP_FLOAT" : Void   // FC1, SCL
{ S7_Optimized_Access := 'TRUE' }
VERSION : 0.1
   VAR_INPUT
      in : Real;
      min : Real;
      max : Real;
   END_VAR
   VAR_OUTPUT
      out : Real;
   END_VAR
BEGIN
   IF #in < #min THEN
       #out := #min;
   ELSIF #in > #max THEN
       #out := #max;
   ELSE
       #out := #in;
   END_IF;
END_FUNCTION

FUNCTION "NumtoBool" : Void   // FC2, LAD
{ S7_Optimized_Access := 'TRUE' }
VERSION : 0.1
   VAR_INPUT
      Input : Real;
   END_VAR
   VAR_OUTPUT
      Output : Array[0..31] of Bool;
   END_VAR
   VAR_TEMP
      val_temp : DInt;
      count : UInt;
   END_VAR
   VAR CONSTANT
      two : Int := 2;
      one : DInt := 1;
   END_VAR
BEGIN

REGION Network 1
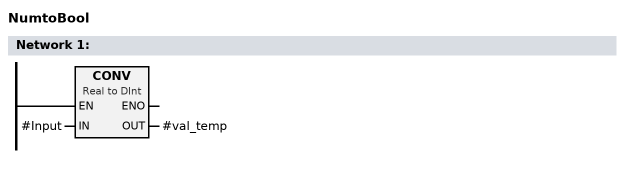
   RUNG wire#powerrail
      { S7_Templates := "[SrcType := Real, DestType := DInt]" } Convert(in := #Input, out => #val_temp)
   END_RUNG
   // the same network as SCL:
   #val_temp := REAL_TO_DINT(#Input);
END_REGION

REGION Network 2 (SCL)

   FOR #count := 0 TO 31 DO
       IF (#val_temp AND SHL(IN:=#one, N:=#count)) <> 0 THEN // Statement section FOR
           #Output[#count] := TRUE;
       ELSE
           #Output[#count] := FALSE;
       END_IF;
   END_FOR;
END_REGION
END_FUNCTION

FUNCTION "cam_zer_rdgs" : Void   // FC3, LAD
{ S7_Optimized_Access := 'TRUE' }
VERSION : 0.1
BEGIN

REGION Network 1 (SCL)
   "Cam".cam_WIDTH := 0;
   "Cam".cam_LENGTH := 0;
   "Cam".cam_Xpos := 0;
   "Cam".cam_Ypos := 0;
   "Cam".cam_Zpos := 0;
   "Cam".cam_DATA := 0;
   "Cam".cam_MAG := 0;
   "Cam".cam_PEAK := 0;
   "Cam".cam_OB_pk := 0;
   "Cam".image_KV := -0;
   "Cam".image_MA := 0;
   "Cam".image_G1 := 0;
   "Cam".image_G2 := 0;
   "Cam".image_BIAS := 0;
   "Cam".image_DIFF := 0;
END_REGION
END_FUNCTION

FUNCTION "ProcCheck" : Void   // FC4, LAD
{ S7_Optimized_Access := 'TRUE' }
VERSION : 0.1
   VAR_INPUT
      inputarray : Array[0..31] of Bool;
   END_VAR
   VAR_OUTPUT
      Result : Bool;
   END_VAR
   VAR_TEMP
      idx : Int;
      out_temp : Bool;
   END_VAR
BEGIN

REGION Network 1 (SCL)
   #out_temp := TRUE;
   FOR #idx := 0 TO 31 DO
       #out_temp := #out_temp AND #inputarray[#idx];
   END_FOR;
   #Result := #out_temp;
END_REGION
END_FUNCTION

FUNCTION "cam_info" : Void   // FC5, LAD
{ S7_Optimized_Access := 'TRUE' }
VERSION : 0.1
BEGIN

REGION Network 1 (SCL)
   "Cam".image_KV := ROUND("pulse".pulse_KV);
   "Cam".image_MA := ROUND("pulse".pulse_MA);
   "Cam".image_G1 := "pulse".pulse_G1;
   "Cam".image_G2 := "pulse".pulse_G2;
   "Cam".image_BIAS := ROUND("BIASDIFF".BIAS);
   "Cam".image_DIFF := ROUND("BIASDIFF".DIFF);
   IF ("Params".stp_PARAMS[7] = FALSE) AND ("Limits".LIMITS_PB[4] = TRUE) THEN
       "Cam".STORE_IMAGE := TRUE;
   ELSE
       "Cam".STORE_IMAGE := FALSE;
   END_IF;
END_REGION
END_FUNCTION

FUNCTION "MIN_MAX" : Void   // FC6, LAD
{ S7_Optimized_Access := 'TRUE' }
VERSION : 0.1
   VAR_INPUT
      TESTVAL : Real;
   END_VAR
   VAR_OUTPUT
      Pass_Fail : Int;
   END_VAR
BEGIN

REGION Network 1 (SCL)
   IF (#TESTVAL >= "StepVals".min) OR (#TESTVAL <= "StepVals".max) THEN
       #Pass_Fail := 1;   //PASS
   ELSE
       #Pass_Fail := -1;  //FAIL
   END_IF;
END_REGION
END_FUNCTION